C05480=1211.778,235.432,-60.754,-177.175,6.527,148.360
C05481=1211.773,235.681,-60.780,-177.172,6.529,148.360
C05482=1211.768,235.930,-60.806,-177.170,6.531,148.360
C05483=1211.764,236.179,-60.832,-177.168,6.533,148.360
C05484=1211.759,236.427,-60.857,-177.165,6.535,148.359
C05485=1211.755,236.676,-60.883,-177.163,6.537,148.359
C05486=1211.751,236.947,-60.912,-177.160,6.540,148.359
C05487=1211.745,237.218,-60.939,-177.157,6.542,148.359
C05488=1211.740,237.490,-60.968,-177.154,6.544,148.358
C05489=1211.736,237.761,-60.997,-177.151,6.546,148.358
C05490=1211.731,238.010,-61.022,-177.148,6.548,148.358
C05491=1211.727,238.258,-61.048,-177.146,6.550,148.358
C05492=1211.722,238.507,-61.074,-177.144,6.552,148.357
C05493=1211.717,238.756,-61.100,-177.141,6.554,148.357
C05494=1211.713,239.004,-61.126,-177.138,6.557,148.357
C05495=1211.709,239.253,-61.152,-177.136,6.559,148.357
C05496=1211.704,239.501,-61.178,-177.133,6.561,148.356
C05497=1211.699,239.751,-61.204,-177.131,6.563,148.356
C05498=1211.695,239.999,-61.230,-177.128,6.565,148.356
C05499=1211.691,240.247,-61.256,-177.126,6.567,148.356
C05500=1211.686,240.496,-61.282,-177.123,6.568,148.355
C05501=1211.682,240.745,-61.308,-177.120,6.571,148.355
C05502=1211.677,240.994,-61.334,-177.118,6.573,148.355
C05503=1211.673,241.242,-61.360,-177.115,6.575,148.355
C05504=1211.668,241.491,-61.387,-177.113,6.577,148.355
C05505=1211.664,241.739,-61.412,-177.110,6.579,148.354
C05506=1211.660,241.987,-61.438,-177.108,6.581,148.354
C05507=1211.655,242.236,-61.465,-177.105,6.583,148.354
C05508=1211.650,242.485,-61.491,-177.102,6.586,148.354
C05509=1211.647,242.733,-61.517,-177.100,6.588,148.353
C05510=1211.642,242.982,-61.543,-177.097,6.590,148.353
C05511=1211.637,243.230,-61.569,-177.095,6.592,148.353
C05512=1211.632,243.479,-61.596,-177.092,6.594,148.352
C05513=1211.628,243.728,-61.622,-177.090,6.596,148.352
C05514=1211.624,243.976,-61.648,-177.088,6.598,148.352
C05515=1211.619,244.225,-61.674,-177.084,6.600,148.352
C05516=1211.615,244.473,-61.701,-177.082,6.602,148.351
C05517=1211.610,244.722,-61.727,-177.080,6.604,148.351
C05518=1211.606,244.971,-61.754,-177.077,6.606,148.351
C05519=1211.602,245.219,-61.779,-177.075,6.609,148.351
C05520=1211.596,245.468,-61.805,-177.072,6.610,148.351
C05521=1211.592,245.716,-61.832,-177.069,6.613,148.350
C05522=1211.588,245.965,-61.858,-177.067,6.615,148.350
C05523=1211.584,246.213,-61.885,-177.064,6.617,148.350
C05524=1211.579,246.462,-61.912,-177.062,6.619,148.350
C05525=1211.575,246.711,-61.937,-177.060,6.621,148.350
C05526=1211.570,246.959,-61.965,-177.057,6.623,148.349
C05527=1211.566,247.208,-61.990,-177.054,6.626,148.349
C05528=1211.561,247.456,-62.017,-177.052,6.628,148.349
C05529=1211.557,247.705,-62.043,-177.049,6.630,148.349
C05530=1211.552,247.954,-62.070,-177.046,6.632,148.348
C05531=1211.548,248.202,-62.097,-177.044,6.634,148.348
C05532=1211.543,248.451,-62.123,-177.041,6.636,148.348
C05533=1211.540,248.699,-62.149,-177.039,6.639,148.348
C05534=1211.535,248.948,-62.176,-177.036,6.641,148.348
C05535=1211.531,249.196,-62.202,-177.034,6.642,148.347
C05536=1211.526,249.445,-62.229,-177.032,6.645,148.347
C05537=1211.521,249.693,-62.255,-177.029,6.646,148.347
C05538=1211.516,249.941,-62.282,-177.026,6.649,148.347
C05539=1211.512,250.190,-62.309,-177.024,6.651,148.346
C05540=1211.508,250.438,-62.335,-177.021,6.653,148.346
C05541=1211.503,250.687,-62.362,-177.019,6.655,148.346
C05542=1211.499,250.935,-62.388,-177.016,6.657,148.346
C05543=1211.494,251.184,-62.415,-177.013,6.660,148.345
C05544=1211.490,251.432,-62.442,-177.011,6.662,148.345
C05545=1211.486,251.682,-62.468,-177.008,6.664,148.345
C05546=1211.481,251.930,-62.495,-177.006,6.666,148.345
C05547=1211.478,252.179,-62.522,-177.003,6.669,148.345
C05548=1211.473,252.427,-62.549,-177.000,6.671,148.344
C05549=1211.468,252.676,-62.576,-176.998,6.673,148.344
C05550=1211.464,252.924,-62.602,-176.996,6.675,148.344
C05551=1211.459,253.173,-62.629,-176.993,6.677,148.344
C05552=1211.455,253.421,-62.656,-176.990,6.680,148.344
C05553=1211.450,253.670,-62.683,-176.988,6.682,148.344
C05554=1211.446,253.918,-62.709,-176.986,6.684,148.343
C05555=1211.441,254.167,-62.736,-176.983,6.686,148.343
C05556=1211.437,254.415,-62.763,-176.981,6.688,148.343
C05557=1211.433,254.664,-62.789,-176.978,6.690,148.343
C05558=1211.428,254.912,-62.816,-176.975,6.693,148.342
C05559=1211.423,255.161,-62.843,-176.973,6.694,148.342
C05560=1211.419,255.409,-62.870,-176.971,6.697,148.342
C05561=1211.415,255.658,-62.897,-176.968,6.699,148.342
C05562=1211.411,255.907,-62.924,-176.965,6.701,148.342
C05563=1211.406,256.155,-62.951,-176.963,6.703,148.341
C05564=1211.401,256.404,-62.978,-176.960,6.705,148.341
C05565=1211.397,256.652,-63.005,-176.957,6.708,148.341
C05566=1211.393,256.900,-63.032,-176.955,6.710,148.341
C05567=1211.388,257.149,-63.059,-176.953,6.712,148.341
C05568=1211.383,257.397,-63.086,-176.950,6.714,148.340
C05569=1211.379,257.646,-63.113,-176.947,6.717,148.340
C05570=1211.375,257.894,-63.140,-176.945,6.719,148.340
C05571=1211.371,258.143,-63.167,-176.942,6.721,148.340
C05572=1211.366,258.391,-63.195,-176.940,6.723,148.340
C05573=1211.362,258.640,-63.222,-176.937,6.726,148.339
C05574=1211.357,258.888,-63.249,-176.935,6.728,148.339
C05575=1211.352,259.137,-63.276,-176.932,6.730,148.339
C05576=1211.349,259.385,-63.302,-176.930,6.732,148.339
C05577=1211.344,259.634,-63.330,-176.927,6.735,148.339
C05578=1211.340,259.883,-63.357,-176.925,6.737,148.339
C05579=1211.335,260.131,-63.384,-176.922,6.739,148.338
C05580=1211.331,260.379,-63.412,-176.920,6.741,148.338
C05581=1211.326,260.627,-63.439,-176.917,6.744,148.338
C05582=1211.321,260.876,-63.466,-176.915,6.746,148.338
C05583=1211.317,261.125,-63.493,-176.912,6.748,148.338
C05584=1211.313,261.374,-63.520,-176.910,6.750,148.337
C05585=1211.308,261.621,-63.548,-176.907,6.753,148.337
C05586=1211.305,261.870,-63.575,-176.904,6.755,148.337
C05587=1211.300,262.118,-63.602,-176.902,6.757,148.337
C05588=1211.296,262.367,-63.629,-176.899,6.760,148.337
C05589=1211.291,262.615,-63.657,-176.897,6.762,148.336
C05590=1211.286,262.888,-63.687,-176.894,6.763,148.336
C05591=1211.281,263.161,-63.716,-176.891,6.766,148.336
C05592=1211.277,263.434,-63.747,-176.888,6.769,148.336
C05593=1211.272,263.706,-63.777,-176.886,6.771,148.336
C05594=1211.268,263.954,-63.804,-176.883,6.774,148.336
C05595=1211.263,264.203,-63.831,-176.881,6.776,148.335
C05596=1211.259,264.452,-63.859,-176.878,6.778,148.335
C05597=1211.254,264.700,-63.887,-176.876,6.780,148.335
C05598=1211.249,264.949,-63.914,-176.873,6.783,148.335
C05599=1211.245,265.197,-63.941,-176.871,6.785,148.335
C05600=1211.241,265.446,-63.970,-176.868,6.787,148.334
C05601=1211.236,265.694,-63.997,-176.865,6.790,148.334
C05602=1211.232,265.942,-64.024,-176.863,6.792,148.334
C05603=1211.227,266.191,-64.051,-176.861,6.794,148.334
C05604=1211.224,266.439,-64.080,-176.857,6.797,148.334
C05605=1211.219,266.688,-64.107,-176.855,6.799,148.334
C05606=1211.215,266.936,-64.134,-176.853,6.801,148.333
C05607=1211.210,267.185,-64.162,-176.850,6.804,148.333
C05608=1211.206,267.433,-64.190,-176.848,6.806,148.333
C05609=1211.201,267.681,-64.217,-176.845,6.808,148.333
C05610=1211.197,267.930,-64.245,-176.843,6.810,148.333
C05611=1211.192,268.179,-64.272,-176.840,6.813,148.333
C05612=1211.188,268.426,-64.300,-176.838,6.815,148.333
C05613=1211.184,268.676,-64.328,-176.835,6.817,148.332
C05614=1211.180,268.923,-64.355,-176.832,6.820,148.332
C05615=1211.175,269.172,-64.383,-176.830,6.822,148.332
C05616=1211.170,269.421,-64.411,-176.828,6.824,148.332
C05617=1211.166,269.669,-64.439,-176.825,6.827,148.332
C05618=1211.161,269.917,-64.466,-176.822,6.829,148.331
C05619=1211.158,270.166,-64.494,-176.820,6.831,148.331
C05620=1211.153,270.414,-64.522,-176.817,6.834,148.331
C05621=1211.148,270.662,-64.550,-176.815,6.836,148.331
C05622=1211.144,270.911,-64.578,-176.812,6.838,148.331
C05623=1211.140,271.159,-64.606,-176.810,6.841,148.331
C05624=1211.135,271.407,-64.633,-176.808,6.843,148.331
C05625=1211.131,271.656,-64.661,-176.805,6.845,148.330
C05626=1211.126,271.904,-64.689,-176.802,6.848,148.330
C05627=1211.122,272.153,-64.717,-176.800,6.850,148.330
C05628=1211.118,272.401,-64.744,-176.797,6.852,148.330
C05629=1211.113,272.649,-64.773,-176.795,6.855,148.330
C05630=1211.109,272.898,-64.801,-176.792,6.857,148.330
C05631=1211.104,273.147,-64.828,-176.790,6.859,148.330
C05632=1211.101,273.395,-64.856,-176.787,6.862,148.329
C05633=1211.096,273.643,-64.884,-176.785,6.864,148.329
C05634=1211.092,273.892,-64.913,-176.782,6.867,148.329
C05635=1211.087,274.140,-64.940,-176.779,6.869,148.329
C05636=1211.082,274.388,-64.969,-176.777,6.871,148.329
C05637=1211.078,274.637,-64.996,-176.775,6.874,148.329
C05638=1211.074,274.885,-65.024,-176.772,6.876,148.328
C05639=1211.070,275.134,-65.053,-176.770,6.878,148.328
C05640=1211.065,275.382,-65.080,-176.767,6.881,148.328
C05641=1211.061,275.630,-65.109,-176.765,6.883,148.328
C05642=1211.056,275.879,-65.137,-176.762,6.885,148.328
C05643=1211.053,276.127,-65.165,-176.759,6.888,148.328
C05644=1211.048,276.375,-65.193,-176.757,6.890,148.328
C05645=1211.044,276.624,-65.222,-176.754,6.893,148.328
C05646=1211.039,276.872,-65.249,-176.752,6.895,148.327
C05647=1211.035,277.121,-65.278,-176.750,6.897,148.327
C05648=1211.031,277.368,-65.306,-176.747,6.900,148.327
C05649=1211.026,277.617,-65.335,-176.744,6.902,148.327
C05650=1211.022,277.865,-65.362,-176.742,6.904,148.327
C05651=1211.018,278.114,-65.391,-176.739,6.907,148.327
C05652=1211.013,278.362,-65.419,-176.737,6.909,148.327
C05653=1211.009,278.611,-65.447,-176.734,6.912,148.327
C05654=1211.004,278.859,-65.475,-176.732,6.914,148.326
C05655=1211.000,279.107,-65.504,-176.730,6.916,148.326
C05656=1210.995,279.356,-65.532,-176.727,6.919,148.326
C05657=1210.991,279.604,-65.560,-176.725,6.922,148.326
C05658=1210.986,279.852,-65.589,-176.722,6.924,148.326
C05659=1210.983,280.101,-65.617,-176.719,6.927,148.326
C05660=1210.978,280.350,-65.645,-176.717,6.929,148.326
C05661=1210.974,280.598,-65.673,-176.714,6.931,148.325
C05662=1210.970,280.846,-65.703,-176.712,6.934,148.325
C05663=1210.965,281.094,-65.730,-176.709,6.937,148.325
C05664=1210.961,281.343,-65.759,-176.707,6.939,148.325
C05665=1210.956,281.591,-65.787,-176.705,6.941,148.325
C05666=1210.952,281.839,-65.816,-176.702,6.944,148.325
C05667=1210.948,282.088,-65.844,-176.699,6.946,148.325
C05668=1210.943,282.336,-65.873,-176.697,6.949,148.325
C05669=1210.939,282.584,-65.902,-176.695,6.951,148.325
C05670=1210.935,282.832,-65.929,-176.692,6.953,148.325
C05671=1210.930,283.081,-65.958,-176.689,6.956,148.324
C05672=1210.927,283.329,-65.987,-176.687,6.958,148.324
C05673=1210.922,283.577,-66.015,-176.684,6.961,148.324
C05674=1210.917,283.826,-66.044,-176.682,6.963,148.324
C05675=1210.913,284.074,-66.072,-176.679,6.966,148.324
C05676=1210.908,284.322,-66.101,-176.677,6.968,148.324
C05677=1210.904,284.571,-66.130,-176.675,6.970,148.324
C05678=1210.900,284.819,-66.158,-176.672,6.973,148.323
C05679=1210.895,285.067,-66.187,-176.670,6.975,148.323
C05680=1210.891,285.316,-66.216,-176.667,6.978,148.323
C05681=1210.887,285.564,-66.245,-176.665,6.980,148.323
C05682=1210.882,285.812,-66.273,-176.662,6.982,148.323
C05683=1210.878,286.061,-66.302,-176.659,6.985,148.323
C05684=1210.874,286.309,-66.330,-176.657,6.988,148.323
C05685=1210.869,286.558,-66.359,-176.655,6.991,148.323
C05686=1210.865,286.806,-66.389,-176.652,6.992,148.323
C05687=1210.861,287.054,-66.416,-176.649,6.995,148.323
C05688=1210.856,287.303,-66.445,-176.647,6.998,148.323
C05689=1210.852,287.551,-66.475,-176.645,7.001,148.323
C05690=1210.847,287.799,-66.503,-176.642,7.003,148.322
C05691=1210.844,288.047,-66.532,-176.640,7.005,148.322
C05692=1210.839,288.296,-66.561,-176.637,7.008,148.322
C05693=1210.834,288.543,-66.590,-176.635,7.010,148.322
C05694=1210.830,288.818,-66.622,-176.632,7.013,148.322
C05695=1210.825,289.093,-66.653,-176.629,7.016,148.322
C05696=1210.821,289.367,-66.686,-176.626,7.019,148.322
C05697=1210.816,289.641,-66.717,-176.624,7.022,148.322
C05698=1210.811,289.888,-66.746,-176.621,7.024,148.321
C05699=1210.807,290.137,-66.775,-176.619,7.026,148.321
C05700=1210.803,290.386,-66.805,-176.616,7.029,148.321
C05701=1210.798,290.635,-66.833,-176.614,7.031,148.321
C05702=1210.793,290.882,-66.862,-176.612,7.034,148.321
C05703=1210.790,291.130,-66.891,-176.609,7.036,148.321
C05704=1210.785,291.379,-66.920,-176.606,7.039,148.321
C05705=1210.781,291.627,-66.950,-176.604,7.041,148.321
C05706=1210.776,291.875,-66.979,-176.601,7.044,148.321
C05707=1210.772,292.124,-67.007,-176.599,7.046,148.321
C05708=1210.768,292.372,-67.037,-176.597,7.049,148.321
C05709=1210.764,292.620,-67.066,-176.594,7.051,148.321
C05710=1210.759,292.868,-67.096,-176.591,7.054,148.321
C05711=1210.755,293.116,-67.123,-176.589,7.057,148.320
C05712=1210.751,293.365,-67.153,-176.587,7.059,148.320
C05713=1210.747,293.613,-67.182,-176.584,7.062,148.320
C05714=1210.743,293.861,-67.212,-176.582,7.064,148.320
C05715=1210.738,294.110,-67.241,-176.579,7.067,148.320
C05716=1210.733,294.358,-67.270,-176.577,7.069,148.320
C05717=1210.729,294.606,-67.299,-176.574,7.072,148.320
C05718=1210.725,294.854,-67.329,-176.572,7.074,148.320
C05719=1210.721,295.102,-67.358,-176.570,7.077,148.320
C05720=1210.716,295.351,-67.387,-176.567,7.079,148.320
C05721=1210.712,295.600,-67.416,-176.565,7.082,148.320
C05722=1210.707,295.847,-67.445,-176.563,7.085,148.320
C05723=1210.703,296.095,-67.475,-176.559,7.087,148.320
C05724=1210.699,296.344,-67.504,-176.557,7.090,148.319
C05725=1210.695,296.592,-67.534,-176.555,7.093,148.319
C05726=1210.691,296.840,-67.563,-176.553,7.095,148.319
C05727=1210.686,297.088,-67.593,-176.550,7.098,148.319
C05728=1210.682,297.337,-67.622,-176.548,7.100,148.319
C05729=1210.678,297.585,-67.651,-176.545,7.103,148.319
C05730=1210.673,297.833,-67.681,-176.543,7.105,148.319
C05731=1210.669,298.081,-67.710,-176.540,7.108,148.319
C05732=1210.665,298.329,-67.739,-176.538,7.110,148.319
C05733=1210.661,298.577,-67.769,-176.535,7.114,148.319
C05734=1210.657,298.826,-67.798,-176.533,7.115,148.319
C05735=1210.652,299.074,-67.828,-176.530,7.118,148.319
C05736=1210.647,299.322,-67.858,-176.528,7.121,148.319
C05737=1210.643,299.571,-67.887,-176.525,7.124,148.319
C05738=1210.639,299.819,-67.917,-176.523,7.126,148.319
C05739=1210.635,300.067,-67.946,-176.521,7.129,148.319
C05740=1210.631,300.316,-67.976,-176.518,7.131,148.319
C05741=1210.627,300.564,-68.005,-176.516,7.134,148.319
C05742=1210.621,300.812,-68.035,-176.514,7.136,148.319
C05743=1210.617,301.060,-68.064,-176.511,7.139,148.319
C05744=1210.613,301.308,-68.094,-176.509,7.142,148.319
C05745=1210.609,301.556,-68.124,-176.506,7.145,148.318
C05746=1210.605,301.804,-68.153,-176.504,7.147,148.318
C05747=1210.600,302.052,-68.183,-176.501,7.150,148.318
C05748=1210.595,302.301,-68.213,-176.499,7.152,148.318
C05749=1210.591,302.549,-68.242,-176.496,7.155,148.318
C05750=1210.587,302.798,-68.272,-176.494,7.157,148.318
C05751=1210.583,303.045,-68.302,-176.492,7.160,148.318
C05752=1210.579,303.293,-68.331,-176.490,7.162,148.318
C05753=1210.574,303.542,-68.361,-176.487,7.166,148.318
C05754=1210.570,303.790,-68.391,-176.485,7.168,148.318
C05755=1210.566,304.038,-68.421,-176.482,7.171,148.318
C05756=1210.561,304.287,-68.451,-176.480,7.173,148.318
C05757=1210.557,304.535,-68.481,-176.477,7.176,148.318
C05758=1210.553,304.782,-68.511,-176.475,7.178,148.318
C05759=1210.549,305.031,-68.540,-176.472,7.181,148.318
C05760=1210.544,305.279,-68.570,-176.470,7.184,148.318
C05761=1210.540,305.528,-68.600,-176.468,7.186,148.318
C05762=1210.536,305.775,-68.630,-176.465,7.189,148.318
C05763=1210.531,306.024,-68.660,-176.463,7.192,148.318
C05764=1210.527,306.271,-68.690,-176.460,7.195,148.318
C05765=1210.523,306.520,-68.720,-176.458,7.197,148.318
C05766=1210.518,306.768,-68.750,-176.455,7.200,148.318
C05767=1210.514,307.016,-68.780,-176.453,7.202,148.318
C05768=1210.510,307.264,-68.809,-176.451,7.205,148.318
C05769=1210.506,307.513,-68.840,-176.448,7.207,148.318
C05770=1210.502,307.761,-68.870,-176.446,7.210,148.318
C05771=1210.497,308.009,-68.901,-176.444,7.213,148.318
C05772=1210.493,308.257,-68.930,-176.441,7.216,148.318
C05773=1210.489,308.506,-68.959,-176.439,7.218,148.318
C05774=1210.484,308.754,-68.990,-176.437,7.221,148.318
C05775=1210.480,309.002,-69.020,-176.434,7.224,148.318
C05776=1210.475,309.250,-69.050,-176.432,7.226,148.318
C05777=1210.472,309.497,-69.081,-176.429,7.229,148.318
C05778=1210.467,309.746,-69.110,-176.427,7.232,148.318
C05779=1210.463,309.994,-69.141,-176.424,7.235,148.318
C05780=1210.459,310.243,-69.171,-176.422,7.237,148.318
C05781=1210.455,310.491,-69.201,-176.420,7.240,148.318
C05782=1210.450,310.739,-69.231,-176.418,7.242,148.318
C05783=1210.446,310.987,-69.262,-176.415,7.246,148.318
C05784=1210.442,311.234,-69.292,-176.413,7.248,148.318
C05785=1210.437,311.483,-69.322,-176.410,7.251,148.318
C05786=1210.433,311.731,-69.352,-176.408,7.254,148.318
C05787=1210.428,311.979,-69.382,-176.406,7.256,148.318
C05788=1210.425,312.228,-69.413,-176.403,7.259,148.318
C05789=1210.420,312.476,-69.443,-176.401,7.262,148.318
C05790=1210.416,312.723,-69.474,-176.399,7.265,148.318
C05791=1210.411,312.972,-69.504,-176.397,7.267,148.318
C05792=1210.408,313.219,-69.534,-176.394,7.270,148.318
C05793=1210.403,313.467,-69.564,-176.392,7.272,148.318
C05794=1210.399,313.716,-69.594,-176.389,7.275,148.318
C05795=1210.395,313.964,-69.625,-176.387,7.278,148.318
C05796=1210.390,314.212,-69.656,-176.385,7.281,148.318
C05797=1210.386,314.460,-69.686,-176.382,7.284,148.318
C05798=1210.381,314.736,-69.720,-176.379,7.287,148.318
C05799=1210.376,315.012,-69.754,-176.377,7.289,148.318
C05800=1210.371,315.289,-69.787,-176.375,7.292,148.318
C05801=1210.368,315.565,-69.821,-176.372,7.295,148.318
C05802=1210.363,315.813,-69.852,-176.370,7.298,148.318
C05803=1210.359,316.061,-69.883,-176.367,7.301,148.318
C05804=1210.355,316.308,-69.913,-176.365,7.304,148.318
C05805=1210.351,316.558,-69.944,-176.362,7.307,148.318
C05806=1210.346,316.806,-69.974,-176.361,7.309,148.318
C05807=1210.342,317.053,-70.005,-176.358,7.312,148.318
C05808=1210.337,317.301,-70.035,-176.356,7.314,148.318
C05809=1210.333,317.550,-70.066,-176.353,7.317,148.318
C05810=1210.330,317.797,-70.097,-176.351,7.320,148.318
C05811=1210.325,318.045,-70.127,-176.349,7.323,148.318
C05812=1210.320,318.293,-70.158,-176.346,7.326,148.318
C05813=1210.317,318.542,-70.189,-176.344,7.328,148.318
C05814=1210.312,318.790,-70.219,-176.342,7.332,148.318
C05815=1210.308,319.038,-70.250,-176.340,7.334,148.318
C05816=1210.303,319.286,-70.281,-176.337,7.337,148.318
C05817=1210.300,319.534,-70.311,-176.335,7.339,148.318
C05818=1210.295,319.782,-70.342,-176.333,7.342,148.318
C05819=1210.291,320.030,-70.373,-176.330,7.345,148.318
C05820=1210.287,320.278,-70.404,-176.328,7.348,148.319
C05821=1210.283,320.526,-70.434,-176.326,7.351,148.319
C05822=1210.278,320.774,-70.465,-176.324,7.353,148.319
C05823=1210.274,321.023,-70.496,-176.321,7.356,148.319
C05824=1210.270,321.271,-70.527,-176.319,7.359,148.319
C05825=1210.266,321.518,-70.557,-176.317,7.362,148.319
C05826=1210.262,321.766,-70.589,-176.314,7.364,148.319
C05827=1210.257,322.014,-70.620,-176.312,7.367,148.319
C05828=1210.253,322.262,-70.650,-176.310,7.370,148.319
C05829=1210.249,322.511,-70.682,-176.308,7.373,148.319
C05830=1210.244,322.759,-70.712,-176.305,7.376,148.319
C05831=1210.240,323.007,-70.743,-176.303,7.378,148.319
C05832=1210.237,323.255,-70.774,-176.301,7.381,148.319
C05833=1210.232,323.503,-70.805,-176.299,7.384,148.319
C05834=1210.227,323.751,-70.836,-176.296,7.387,148.319
C05835=1210.223,323.999,-70.867,-176.294,7.390,148.319
C05836=1210.219,324.247,-70.899,-176.292,7.392,148.319
C05837=1210.215,324.495,-70.930,-176.290,7.396,148.320
C05838=1210.211,324.743,-70.960,-176.287,7.398,148.319
C05839=1210.206,324.991,-70.991,-176.285,7.401,148.319
C05840=1210.203,325.239,-71.022,-176.283,7.403,148.320
C05841=1210.198,325.487,-71.053,-176.280,7.406,148.320
C05842=1210.194,325.735,-71.084,-176.278,7.410,148.320
C05843=1210.190,325.983,-71.116,-176.276,7.412,148.320
C05844=1210.186,326.231,-71.147,-176.274,7.415,148.320
C05845=1210.181,326.479,-71.178,-176.272,7.417,148.320
C05846=1210.177,326.727,-71.209,-176.269,7.420,148.320
C05847=1210.173,326.975,-71.240,-176.267,7.423,148.320
C05848=1210.168,327.223,-71.271,-176.265,7.426,148.320
C05849=1210.165,327.471,-71.303,-176.263,7.429,148.320
C05850=1210.160,327.719,-71.334,-176.260,7.432,148.320
C05851=1210.156,327.967,-71.366,-176.258,7.435,148.321
C05852=1210.152,328.215,-71.396,-176.256,7.437,148.321
C05853=1210.147,328.463,-71.428,-176.254,7.440,148.321
C05854=1210.143,328.711,-71.459,-176.252,7.443,148.321
C05855=1210.139,328.959,-71.490,-176.250,7.446,148.321
C05856=1210.135,329.207,-71.522,-176.247,7.449,148.321
C05857=1210.130,329.455,-71.552,-176.245,7.452,148.321
C05858=1210.127,329.703,-71.584,-176.243,7.455,148.321
C05859=1210.122,329.951,-71.615,-176.241,7.457,148.321
C05860=1210.118,330.199,-71.647,-176.238,7.460,148.321
C05861=1210.114,330.447,-71.678,-176.237,7.463,148.321
C05862=1210.110,330.695,-71.709,-176.234,7.466,148.321
C05863=1210.106,330.943,-71.741,-176.232,7.469,148.322
C05864=1210.102,331.191,-71.772,-176.230,7.472,148.322
C05865=1210.097,331.439,-71.804,-176.227,7.475,148.322
C05866=1210.093,331.688,-71.835,-176.226,7.477,148.322
C05867=1210.088,331.935,-71.867,-176.223,7.480,148.322
C05868=1210.085,332.183,-71.898,-176.221,7.483,148.322
C05869=1210.080,332.431,-71.929,-176.219,7.486,148.322
C05870=1210.076,332.679,-71.961,-176.217,7.489,148.322
C05871=1210.072,332.926,-71.993,-176.215,7.492,148.323
C05872=1210.068,333.175,-72.024,-176.212,7.495,148.323
C05873=1210.064,333.423,-72.056,-176.211,7.497,148.323
C05874=1210.059,333.671,-72.088,-176.208,7.500,148.323
C05875=1210.055,333.919,-72.119,-176.206,7.503,148.323
C05876=1210.051,334.167,-72.150,-176.204,7.506,148.323
C05877=1210.047,334.415,-72.182,-176.201,7.509,148.323
C05878=1210.042,334.662,-72.214,-176.200,7.512,148.323
C05879=1210.038,334.911,-72.245,-176.198,7.515,148.324
C05880=1210.034,335.158,-72.277,-176.195,7.517,148.324
C05881=1210.030,335.406,-72.309,-176.193,7.521,148.324
C05882=1210.026,335.654,-72.340,-176.192,7.523,148.324
C05883=1210.021,335.903,-72.372,-176.189,7.526,148.324
C05884=1210.017,336.151,-72.404,-176.187,7.529,148.324
C05885=1210.013,336.398,-72.435,-176.185,7.532,148.324
C05886=1210.009,336.646,-72.467,-176.182,7.535,148.324
C05887=1210.005,336.894,-72.499,-176.181,7.537,148.325
C05888=1210.001,337.142,-72.531,-176.178,7.541,148.325
C05889=1209.997,337.390,-72.563,-176.177,7.543,148.325
C05890=1209.992,337.639,-72.594,-176.174,7.546,148.325
C05891=1209.988,337.886,-72.626,-176.172,7.549,148.325
C05892=1209.984,338.134,-72.658,-176.170,7.552,148.325
C05893=1209.980,338.382,-72.689,-176.168,7.555,148.325
C05894=1209.975,338.630,-72.722,-176.166,7.558,148.326
C05895=1209.972,338.878,-72.754,-176.164,7.561,148.326
C05896=1209.967,339.125,-72.785,-176.162,7.564,148.326
C05897=1209.963,339.374,-72.817,-176.160,7.567,148.326
C05898=1209.959,339.622,-72.849,-176.158,7.569,148.326
C05899=1209.955,339.869,-72.881,-176.156,7.573,148.326
C05900=1209.951,340.117,-72.913,-176.153,7.576,148.327
C05901=1209.947,340.365,-72.945,-176.152,7.578,148.327
C05902=1209.942,340.643,-72.981,-176.149,7.581,148.327
C05903=1209.937,340.921,-73.016,-176.147,7.585,148.327
C05904=1209.933,341.200,-73.053,-176.145,7.588,148.327
C05905=1209.928,341.478,-73.089,-176.142,7.592,148.327
C05906=1209.924,341.726,-73.121,-176.140,7.595,148.328
C05907=1209.919,341.973,-73.153,-176.139,7.597,148.328
C05908=1209.915,342.222,-73.185,-176.136,7.600,148.328
C05909=1209.911,342.470,-73.217,-176.134,7.603,148.328
C05910=1209.906,342.717,-73.249,-176.132,7.606,148.328
C05911=1209.903,342.965,-73.280,-176.130,7.609,148.328
C05912=1209.899,343.213,-73.314,-176.128,7.612,148.329
C05913=1209.894,343.460,-73.345,-176.127,7.615,148.329
C05914=1209.890,343.709,-73.378,-176.124,7.618,148.329
C05915=1209.886,343.957,-73.409,-176.122,7.621,148.329
C05916=1209.882,344.205,-73.442,-176.120,7.624,148.329
C05917=1209.877,344.452,-73.473,-176.118,7.627,148.329
C05918=1209.873,344.700,-73.506,-176.116,7.629,148.330
C05919=1209.869,344.948,-73.538,-176.114,7.633,148.330
C05920=1209.865,345.196,-73.571,-176.112,7.635,148.330
C05921=1209.861,345.444,-73.602,-176.110,7.639,148.330
C05922=1209.857,345.692,-73.635,-176.108,7.641,148.330
C05923=1209.853,345.940,-73.667,-176.106,7.645,148.331
C05924=1209.848,346.188,-73.700,-176.105,7.647,148.331
C05925=1209.843,346.436,-73.732,-176.102,7.650,148.331
C05926=1209.840,346.683,-73.764,-176.101,7.653,148.331
C05927=1209.836,346.931,-73.797,-176.098,7.656,148.331
C05928=1209.832,347.179,-73.829,-176.096,7.660,148.332
C05929=1209.828,347.427,-73.862,-176.095,7.662,148.332
C05930=1209.823,347.674,-73.893,-176.092,7.665,148.332
C05931=1209.819,347.923,-73.926,-176.091,7.668,148.332
C05932=1209.815,348.171,-73.959,-176.089,7.671,148.332
C05933=1209.811,348.419,-73.991,-176.087,7.674,148.333
C05934=1209.807,348.666,-74.024,-176.085,7.677,148.333
C05935=1209.802,348.914,-74.056,-176.083,7.680,148.333
C05936=1209.798,349.162,-74.088,-176.081,7.683,148.333
C05937=1209.794,349.410,-74.121,-176.079,7.686,148.333
C05938=1209.790,349.658,-74.153,-176.077,7.689,148.334
C05939=1209.786,349.905,-74.186,-176.076,7.692,148.334
C05940=1209.781,350.153,-74.218,-176.074,7.695,148.334
C05941=1209.778,350.401,-74.251,-176.072,7.698,148.334
C05942=1209.773,350.649,-74.283,-176.070,7.701,148.335
C05943=1209.769,350.897,-74.316,-176.068,7.703,148.335
C05944=1209.766,351.145,-74.348,-176.066,7.707,148.335
C05945=1209.761,351.392,-74.381,-176.064,7.709,148.335
C05946=1209.757,351.641,-74.414,-176.062,7.713,148.336
C05947=1209.752,351.888,-74.446,-176.061,7.715,148.336
C05948=1209.748,352.136,-74.478,-176.059,7.719,148.336
C05949=1209.744,352.384,-74.511,-176.057,7.721,148.336
C05950=1209.740,352.632,-74.544,-176.055,7.725,148.337
C05951=1209.737,352.879,-74.576,-176.053,7.727,148.337
C05952=1209.732,353.127,-74.610,-176.051,7.731,148.337
C05953=1209.728,353.375,-74.642,-176.050,7.733,148.337
C05954=1209.724,353.623,-74.675,-176.047,7.737,148.338
C05955=1209.719,353.871,-74.708,-176.046,7.739,148.338
C05956=1209.715,354.118,-74.740,-176.044,7.743,148.338
C05957=1209.711,354.366,-74.773,-176.042,7.745,148.338
C05958=1209.707,354.614,-74.805,-176.040,7.749,148.339
C05959=1209.703,354.862,-74.839,-176.039,7.751,148.339
C05960=1209.699,355.109,-74.871,-176.037,7.755,148.339
C05961=1209.695,355.358,-74.904,-176.035,7.757,148.339
C05962=1209.691,355.606,-74.937,-176.033,7.761,148.340
C05963=1209.687,355.853,-74.970,-176.031,7.763,148.340
C05964=1209.682,356.101,-75.003,-176.030,7.767,148.340
C05965=1209.678,356.349,-75.035,-176.028,7.769,148.340
C05966=1209.675,356.597,-75.068,-176.026,7.773,148.341
C05967=1209.670,356.844,-75.101,-176.024,7.776,148.341
C05968=1209.666,357.092,-75.134,-176.022,7.779,148.341
C05969=1209.662,357.341,-75.167,-176.021,7.781,148.341
C05970=1209.658,357.588,-75.200,-176.019,7.785,148.342
C05971=1209.654,357.836,-75.233,-176.017,7.788,148.342
C05972=1209.649,358.084,-75.266,-176.015,7.791,148.343
C05973=1209.646,358.331,-75.299,-176.014,7.794,148.343
C05974=1209.642,358.580,-75.331,-176.012,7.797,148.343
C05975=1209.637,358.827,-75.364,-176.010,7.800,148.343
C05976=1209.633,359.074,-75.397,-176.008,7.803,148.344
C05977=1209.629,359.322,-75.430,-176.007,7.806,148.344
C05978=1209.624,359.570,-75.463,-176.005,7.809,148.344
C05979=1209.620,359.817,-75.497,-176.003,7.812,148.344
C05980=1209.616,360.065,-75.530,-176.002,7.815,148.345
C05981=1209.613,360.314,-75.563,-176.000,7.818,148.345
C05982=1209.608,360.561,-75.596,-175.999,7.821,148.345
C05983=1209.604,360.810,-75.629,-175.996,7.824,148.346
C05984=1209.600,361.057,-75.662,-175.995,7.827,148.346
C05985=1209.596,361.305,-75.695,-175.993,7.830,148.346
C05986=1209.592,361.553,-75.728,-175.992,7.833,148.347
C05987=1209.587,361.801,-75.762,-175.990,7.836,148.347
C05988=1209.584,362.048,-75.794,-175.988,7.839,148.347
C05989=1209.580,362.296,-75.827,-175.987,7.842,148.348
C05990=1209.576,362.543,-75.860,-175.985,7.846,148.348
C05991=1209.572,362.791,-75.894,-175.984,7.848,148.348
C05992=1209.567,363.039,-75.927,-175.982,7.851,148.348
C05993=1209.563,363.287,-75.960,-175.980,7.855,148.349
C05994=1209.558,363.535,-75.994,-175.979,7.857,148.349
C05995=1209.555,363.782,-76.027,-175.977,7.861,148.350
C05996=1209.551,364.030,-76.061,-175.976,7.863,148.350
C05997=1209.546,364.277,-76.094,-175.974,7.866,148.350
C05998=1209.542,364.525,-76.127,-175.972,7.870,148.351
C05999=1209.538,364.773,-76.160,-175.971,7.872,148.351
C06000=1209.535,365.021,-76.194,-175.969,7.875,148.351
C06001=1209.530,365.269,-76.227,-175.968,7.879,148.352
C06002=1209.526,365.517,-76.260,-175.966,7.881,148.352
C06003=1209.522,365.764,-76.293,-175.965,7.884,148.352
C06004=1209.518,366.011,-76.327,-175.963,7.888,148.353
C06005=1209.514,366.259,-76.360,-175.962,7.890,148.353
C06006=1209.509,366.540,-76.398,-175.960,7.894,148.353
C06007=1209.505,366.820,-76.435,-175.958,7.897,148.354
C06008=1209.501,367.100,-76.473,-175.957,7.900,148.354
C06009=1209.495,367.380,-76.511,-175.955,7.904,148.354
C06010=1209.492,367.629,-76.545,-175.954,7.907,148.355
C06011=1209.488,367.876,-76.578,-175.952,7.910,148.355
C06012=1209.483,368.124,-76.611,-175.951,7.913,148.356
C06013=1209.480,368.371,-76.645,-175.949,7.916,148.356
C06014=1209.475,368.619,-76.679,-175.947,7.919,148.356
C06015=1209.471,368.867,-76.712,-175.946,7.922,148.357
C06016=1209.466,369.115,-76.745,-175.945,7.925,148.357
C06017=1209.463,369.362,-76.779,-175.944,7.928,148.358
C06018=1209.459,369.610,-76.813,-175.942,7.931,148.358
C06019=1209.455,369.858,-76.846,-175.940,7.934,148.358
C06020=1209.450,370.105,-76.880,-175.939,7.937,148.359
C06021=1209.446,370.353,-76.913,-175.938,7.940,148.359
C06022=1209.442,370.601,-76.947,-175.936,7.943,148.359
C06023=1209.438,370.848,-76.980,-175.935,7.946,148.360
C06024=1209.435,371.096,-77.014,-175.934,7.949,148.360
C06025=1209.430,371.344,-77.048,-175.933,7.952,148.361
C06026=1209.426,371.592,-77.082,-175.931,7.954,148.361
C06027=1209.422,371.839,-77.115,-175.930,7.958,148.361
C06028=1209.418,372.087,-77.148,-175.928,7.961,148.362
C06029=1209.414,372.335,-77.183,-175.927,7.964,148.362
C06030=1209.410,372.583,-77.216,-175.926,7.966,148.363
C06031=1209.406,372.830,-77.250,-175.925,7.969,148.363
C06032=1209.402,373.078,-77.283,-175.923,7.973,148.363
C06033=1209.397,373.325,-77.317,-175.922,7.976,148.364
C06034=1209.393,373.574,-77.351,-175.921,7.979,148.364
C06035=1209.390,373.821,-77.385,-175.919,7.981,148.365
C06036=1209.385,374.069,-77.418,-175.918,7.984,148.365
C06037=1209.381,374.316,-77.452,-175.917,7.987,148.365
C06038=1209.377,374.564,-77.486,-175.916,7.990,148.366
C06039=1209.373,374.812,-77.520,-175.914,7.993,148.366
C06040=1209.369,375.059,-77.554,-175.913,7.996,148.367
C06041=1209.365,375.307,-77.587,-175.912,7.999,148.367
C06042=1209.361,375.554,-77.621,-175.911,8.002,148.368
C06043=1209.357,375.802,-77.655,-175.910,8.005,148.368
C06044=1209.353,376.050,-77.689,-175.909,8.008,148.368
C06045=1209.349,376.297,-77.722,-175.907,8.011,148.369
C06046=1209.344,376.545,-77.756,-175.906,8.013,148.369
C06047=1209.341,376.793,-77.790,-175.905,8.016,148.370
C06048=1209.336,377.041,-77.824,-175.904,8.019,148.370
C06049=1209.332,377.288,-77.858,-175.903,8.022,148.370
C06050=1209.328,377.535,-77.892,-175.902,8.025,148.371
C06051=1209.324,377.784,-77.926,-175.901,8.028,148.371
C06052=1209.320,378.031,-77.960,-175.899,8.031,148.372
C06053=1209.316,378.279,-77.993,-175.898,8.033,148.372
C06054=1209.311,378.526,-78.027,-175.897,8.037,148.373
C06055=1209.308,378.774,-78.062,-175.896,8.039,148.373
C06056=1209.303,379.022,-78.095,-175.895,8.042,148.373
C06057=1209.299,379.269,-78.129,-175.894,8.045,148.374
C06058=1209.295,379.517,-78.164,-175.893,8.048,148.374
C06059=1209.291,379.765,-78.197,-175.892,8.051,148.375
C06060=1209.287,380.012,-78.231,-175.891,8.054,148.375
C06061=1209.283,380.260,-78.266,-175.889,8.056,148.376
C06062=1209.279,380.508,-78.299,-175.889,8.060,148.376
C06063=1209.275,380.755,-78.334,-175.888,8.062,148.377
C06064=1209.271,381.003,-78.368,-175.886,8.065,148.377
C06065=1209.267,381.251,-78.402,-175.886,8.068,148.378
C06066=1209.263,381.498,-78.436,-175.884,8.071,148.378
C06067=1209.258,381.746,-78.470,-175.883,8.074,148.378
C06068=1209.255,381.994,-78.504,-175.882,8.077,148.379
C06069=1209.251,382.241,-78.537,-175.881,8.080,148.379
C06070=1209.246,382.489,-78.572,-175.880,8.083,148.380
C06071=1209.243,382.737,-78.606,-175.880,8.085,148.380
C06072=1209.239,382.984,-78.641,-175.879,8.088,148.381
C06073=1209.235,383.231,-78.674,-175.878,8.091,148.381
C06074=1209.230,383.479,-78.708,-175.877,8.094,148.382
C06075=1209.227,383.727,-78.742,-175.875,8.096,148.382
C06076=1209.222,383.974,-78.777,-175.875,8.100,148.383
C06077=1209.218,384.223,-78.812,-175.873,8.102,148.383
C06078=1209.214,384.470,-78.846,-175.873,8.105,148.384
C06079=1209.209,384.718,-78.879,-175.872,8.108,148.384
C06080=1209.206,384.965,-78.914,-175.871,8.111,148.385
C06081=1209.202,385.213,-78.948,-175.870,8.113,148.385
C06082=1209.198,385.460,-78.982,-175.869,8.117,148.386
C06083=1209.194,385.708,-79.017,-175.869,8.119,148.386
C06084=1209.190,385.955,-79.051,-175.867,8.121,148.386
C06085=1209.185,386.203,-79.085,-175.867,8.124,148.387
C06086=1209.182,386.450,-79.119,-175.866,8.127,148.387
C06087=1209.177,386.699,-79.153,-175.865,8.130,148.388
C06088=1209.173,386.946,-79.188,-175.864,8.132,148.388
C06089=1209.169,387.194,-79.222,-175.863,8.135,148.389
C06090=1209.165,387.441,-79.256,-175.862,8.138,148.389
C06091=1209.162,387.689,-79.290,-175.862,8.141,148.390
C06092=1209.157,387.936,-79.325,-175.861,8.143,148.390
C06093=1209.153,388.183,-79.359,-175.860,8.146,148.391
C06094=1209.149,388.432,-79.394,-175.860,8.149,148.391
C06095=1209.145,388.679,-79.428,-175.859,8.151,148.392
C06096=1209.141,388.927,-79.462,-175.858,8.155,148.392
C06097=1209.137,389.174,-79.497,-175.857,8.157,148.393
C06098=1209.133,389.421,-79.531,-175.856,8.160,148.393
C06099=1209.129,389.669,-79.566,-175.855,8.162,148.394
C06100=1209.125,389.917,-79.600,-175.855,8.165,148.394
C06101=1209.121,390.165,-79.634,-175.854,8.168,148.394
C06102=1209.117,390.412,-79.669,-175.853,8.171,148.395
C06103=1209.112,390.660,-79.703,-175.853,8.173,148.396
C06104=1209.109,390.907,-79.737,-175.852,8.176,148.396
C06105=1209.104,391.155,-79.772,-175.851,8.179,148.397
C06106=1209.100,391.403,-79.807,-175.850,8.181,148.397
C06107=1209.097,391.650,-79.841,-175.849,8.184,148.398
C06108=1209.093,391.898,-79.875,-175.849,8.186,148.398
C06109=1209.089,392.145,-79.909,-175.848,8.189,148.398
C06110=1209.084,392.428,-79.949,-175.847,8.192,148.399
C06111=1209.079,392.710,-79.988,-175.846,8.195,148.400
C06112=1209.075,392.992,-80.028,-175.846,8.198,148.400
C06113=1209.070,393.275,-80.067,-175.846,8.201,148.401
C06114=1209.066,393.523,-80.101,-175.844,8.203,148.401
C06115=1209.062,393.770,-80.137,-175.844,8.206,148.402
C06116=1209.058,394.017,-80.171,-175.843,8.209,148.402
C06117=1209.054,394.265,-80.205,-175.843,8.211,148.403
C06118=1209.050,394.513,-80.240,-175.842,8.214,148.403
C06119=1209.045,394.760,-80.274,-175.841,8.216,148.404
C06120=1209.042,395.008,-80.309,-175.841,8.219,148.404
C06121=1209.037,395.255,-80.343,-175.840,8.221,148.405
C06122=1209.033,395.504,-80.378,-175.839,8.224,148.405
C06123=1209.030,395.750,-80.413,-175.839,8.226,148.406
C06124=1209.026,395.998,-80.447,-175.838,8.229,148.406
C06125=1209.021,396.246,-80.482,-175.837,8.231,148.407
C06126=1209.017,396.494,-80.517,-175.837,8.235,148.407
C06127=1209.014,396.741,-80.551,-175.837,8.237,148.408
C06128=1209.010,396.988,-80.586,-175.836,8.239,148.408
C06129=1209.005,397.236,-80.621,-175.835,8.242,148.409
C06130=1209.001,397.484,-80.655,-175.835,8.244,148.409
C06131=1208.998,397.731,-80.689,-175.834,8.247,148.410
C06132=1208.994,397.979,-80.724,-175.833,8.249,148.410
C06133=1208.989,398.226,-80.759,-175.833,8.251,148.411
C06134=1208.985,398.474,-80.794,-175.832,8.255,148.411
C06135=1208.981,398.721,-80.829,-175.832,8.257,148.412
C06136=1208.978,398.969,-80.863,-175.832,8.259,148.412
C06137=1208.973,399.216,-80.898,-175.831,8.262,148.413
C06138=1208.969,399.464,-80.933,-175.830,8.264,148.413
C06139=1208.965,399.712,-80.967,-175.830,8.266,148.414
C06140=1208.962,399.959,-81.002,-175.829,8.269,148.414
C06141=1208.957,400.206,-81.037,-175.829,8.271,148.415
C06142=1208.953,400.454,-81.072,-175.828,8.274,148.415
C06143=1208.949,400.702,-81.106,-175.828,8.277,148.416
C06144=1208.945,400.950,-81.141,-175.827,8.279,148.416
C06145=1208.941,401.196,-81.175,-175.827,8.281,148.417
C06146=1208.937,401.444,-81.210,-175.826,8.284,148.417
C06147=1208.933,401.692,-81.245,-175.826,8.286,148.418
C06148=1208.929,401.939,-81.280,-175.825,8.288,148.418
C06149=1208.924,402.187,-81.315,-175.825,8.290,148.419
C06150=1208.921,402.435,-81.350,-175.824,8.294,148.419
C06151=1208.917,402.681,-81.384,-175.823,8.296,148.419
C06152=1208.913,402.929,-81.419,-175.823,8.298,148.420
C06153=1208.908,403.177,-81.453,-175.823,8.300,148.421
C06154=1208.905,403.424,-81.489,-175.822,8.303,148.421
C06155=1208.900,403.672,-81.523,-175.822,8.305,148.421
C06156=1208.896,403.920,-81.558,-175.821,8.307,148.422
C06157=1208.892,404.167,-81.593,-175.821,8.310,148.422
C06158=1208.889,404.415,-81.628,-175.821,8.312,148.423
C06159=1208.885,404.662,-81.663,-175.820,8.315,148.423
C06160=1208.881,404.909,-81.698,-175.820,8.317,148.424
C06161=1208.877,405.158,-81.733,-175.819,8.319,148.424
C06162=1208.872,405.404,-81.768,-175.819,8.321,148.425
C06163=1208.868,405.653,-81.803,-175.818,8.324,148.425
C06164=1208.864,405.899,-81.838,-175.818,8.327,148.426
C06165=1208.860,406.147,-81.873,-175.817,8.329,148.426
C06166=1208.856,406.395,-81.906,-175.817,8.331,148.427
C06167=1208.853,406.642,-81.942,-175.817,8.333,148.427
C06168=1208.849,406.890,-81.977,-175.816,8.335,148.428
C06169=1208.844,407.137,-82.012,-175.816,8.337,148.428
C06170=1208.840,407.385,-82.047,-175.816,8.340,148.429
C06171=1208.836,407.632,-82.082,-175.815,8.342,148.429
C06172=1208.832,407.880,-82.117,-175.814,8.345,148.430
C06173=1208.828,408.127,-82.151,-175.814,8.347,148.430
C06174=1208.824,408.375,-82.187,-175.813,8.349,148.431
C06175=1208.820,408.623,-82.222,-175.813,8.351,148.431
C06176=1208.816,408.870,-82.257,-175.813,8.354,148.432
C06177=1208.812,409.118,-82.291,-175.813,8.356,148.432
C06178=1208.808,409.364,-82.326,-175.812,8.358,148.432
C06179=1208.804,409.613,-82.361,-175.812,8.360,148.433
C06180=1208.801,409.860,-82.397,-175.812,8.362,148.434
C06181=1208.796,410.107,-82.431,-175.811,8.364,148.434
C06182=1208.792,410.355,-82.467,-175.811,8.367,148.434
C06183=1208.788,410.602,-82.501,-175.810,8.370,148.435
C06184=1208.784,410.850,-82.537,-175.809,8.372,148.435
C06185=1208.780,411.098,-82.572,-175.809,8.374,148.436
C06186=1208.776,411.345,-82.607,-175.809,8.376,148.436
C06187=1208.772,411.593,-82.642,-175.808,8.378,148.437
C06188=1208.768,411.840,-82.677,-175.808,8.380,148.437
C06189=1208.764,412.087,-82.712,-175.808,8.383,148.438
C06190=1208.760,412.335,-82.747,-175.807,8.385,148.438
C06191=1208.756,412.582,-82.782,-175.807,8.387,148.439
C06192=1208.752,412.830,-82.817,-175.807,8.389,148.439
C06193=1208.748,413.077,-82.852,-175.806,8.391,148.440
C06194=1208.744,413.325,-82.887,-175.806,8.393,148.440
C06195=1208.740,413.573,-82.923,-175.805,8.396,148.441
C06196=1208.736,413.820,-82.958,-175.805,8.398,148.441
C06197=1208.732,414.068,-82.993,-175.805,8.400,148.441
C06198=1208.728,414.315,-83.028,-175.804,8.402,148.442
C06199=1208.723,414.563,-83.063,-175.804,8.404,148.442
C06200=1208.720,414.810,-83.098,-175.804,8.406,148.443
C06201=1208.715,415.057,-83.133,-175.803,8.409,148.443
C06202=1208.712,415.305,-83.168,-175.803,8.411,148.444
C06203=1208.708,415.552,-83.204,-175.802,8.413,148.444
C06204=1208.703,415.800,-83.238,-175.802,8.415,148.445
C06205=1208.700,416.047,-83.274,-175.802,8.416,148.445
C06206=1208.695,416.309,-83.311,-175.801,8.419,148.446
C06207=1208.692,416.571,-83.348,-175.801,8.421,148.446
C06208=1208.690,416.833,-83.385,-175.800,8.424,148.447
C06209=1208.692,417.093,-83.422,-175.800,8.426,148.447
C06210=1208.270,417.094,-83.458,-175.803,8.436,148.451
C06211=1208.269,416.830,-83.421,-175.804,8.434,148.450
C06212=1208.270,416.565,-83.385,-175.804,8.432,148.450
C06213=1208.274,416.301,-83.347,-175.805,8.430,148.449
C06214=1208.278,416.037,-83.309,-175.805,8.427,148.449
C06215=1208.282,415.789,-83.274,-175.805,8.426,148.448
C06216=1208.286,415.541,-83.239,-175.806,8.424,148.448
C06217=1208.290,415.295,-83.203,-175.806,8.421,148.447
C06218=1208.294,415.046,-83.168,-175.806,8.419,148.447
C06219=1208.298,414.799,-83.133,-175.807,8.417,148.447
C06220=1208.302,414.551,-83.098,-175.807,8.415,148.446
C06221=1208.306,414.304,-83.063,-175.807,8.413,148.446
C06222=1208.310,414.057,-83.028,-175.808,8.411,148.445
C06223=1208.314,413.809,-82.993,-175.808,8.408,148.445
C06224=1208.318,413.562,-82.957,-175.808,8.406,148.444
C06225=1208.323,413.314,-82.923,-175.809,8.404,148.444
C06226=1208.326,413.067,-82.887,-175.809,8.402,148.443
C06227=1208.330,412.819,-82.852,-175.809,8.400,148.443
C06228=1208.334,412.572,-82.817,-175.810,8.398,148.442
C06229=1208.338,412.324,-82.782,-175.810,8.395,148.442
C06230=1208.343,412.077,-82.747,-175.811,8.393,148.441
C06231=1208.346,411.829,-82.712,-175.811,8.391,148.441
C06232=1208.350,411.581,-82.677,-175.811,8.389,148.440
C06233=1208.355,411.334,-82.642,-175.812,8.387,148.440
C06234=1208.359,411.086,-82.607,-175.812,8.385,148.440
C06235=1208.363,410.839,-82.572,-175.812,8.382,148.439
C06236=1208.366,410.592,-82.536,-175.813,8.380,148.439
C06237=1208.370,410.344,-82.501,-175.813,8.378,148.438
C06238=1208.375,410.097,-82.466,-175.814,8.375,148.438
C06239=1208.379,409.849,-82.431,-175.814,8.373,148.437
C06240=1208.383,409.602,-82.396,-175.815,8.370,148.437
C06241=1208.386,409.354,-82.362,-175.815,8.368,148.436
C06242=1208.390,409.107,-82.326,-175.815,8.366,148.436
C06243=1208.394,408.859,-82.292,-175.816,8.364,148.435
C06244=1208.398,408.612,-82.256,-175.816,8.362,148.435
C06245=1208.403,408.364,-82.222,-175.817,8.360,148.434
C06246=1208.406,408.117,-82.186,-175.817,8.357,148.434
C06247=1208.410,407.869,-82.152,-175.817,8.355,148.433
C06248=1208.415,407.621,-82.117,-175.818,8.353,148.433
C06249=1208.418,407.374,-82.082,-175.818,8.350,148.432
C06250=1208.423,407.127,-82.047,-175.819,8.348,148.432
C06251=1208.427,406.879,-82.012,-175.819,8.346,148.431
C06252=1208.431,406.632,-81.977,-175.819,8.344,148.431
C06253=1208.434,406.384,-81.942,-175.820,8.341,148.430
C06254=1208.438,406.136,-81.907,-175.820,8.339,148.430
C06255=1208.442,405.890,-81.872,-175.821,8.337,148.429
C06256=1208.446,405.641,-81.837,-175.821,8.335,148.429
C06257=1208.451,405.394,-81.803,-175.822,8.332,148.429
C06258=1208.455,405.146,-81.767,-175.822,8.330,148.428
C06259=1208.459,404.899,-81.733,-175.822,8.327,148.427
C06260=1208.463,404.652,-81.697,-175.823,8.325,148.427
C06261=1208.467,404.403,-81.662,-175.823,8.323,148.427
C06262=1208.471,404.156,-81.629,-175.824,8.320,148.426
C06263=1208.474,403.909,-81.593,-175.824,8.318,148.425
C06264=1208.479,403.661,-81.558,-175.825,8.316,148.425
C06265=1208.483,403.414,-81.523,-175.825,8.314,148.425
C06266=1208.487,403.166,-81.488,-175.825,8.311,148.424
C06267=1208.491,402.918,-81.454,-175.826,8.308,148.423
C06268=1208.495,402.672,-81.418,-175.827,8.306,148.423
C06269=1208.499,402.424,-81.384,-175.827,8.304,148.423
C06270=1208.503,402.176,-81.350,-175.827,8.302,148.422
C06271=1208.507,401.929,-81.314,-175.828,8.299,148.422
C06272=1208.511,401.681,-81.280,-175.829,8.297,148.421
C06273=1208.515,401.433,-81.245,-175.829,8.294,148.421
C06274=1208.519,401.186,-81.209,-175.829,8.292,148.420
C06275=1208.523,400.939,-81.175,-175.830,8.289,148.420
C06276=1208.527,400.691,-81.141,-175.830,8.287,148.419
C06277=1208.531,400.444,-81.105,-175.831,8.285,148.419
C06278=1208.535,400.196,-81.071,-175.832,8.282,148.418
C06279=1208.540,399.948,-81.036,-175.832,8.280,148.418
C06280=1208.543,399.700,-81.002,-175.832,8.277,148.417
C06281=1208.547,399.454,-80.967,-175.833,8.274,148.417
C06282=1208.551,399.205,-80.932,-175.834,8.272,148.416
C06283=1208.556,398.958,-80.897,-175.834,8.270,148.416
C06284=1208.560,398.710,-80.863,-175.835,8.267,148.415
C06285=1208.563,398.463,-80.828,-175.835,8.265,148.415
C06286=1208.567,398.215,-80.793,-175.836,8.263,148.414
C06287=1208.572,397.968,-80.759,-175.836,8.260,148.414
C06288=1208.576,397.720,-80.724,-175.837,8.258,148.413
C06289=1208.579,397.473,-80.689,-175.838,8.254,148.413
C06290=1208.583,397.225,-80.654,-175.838,8.252,148.412
C06291=1208.588,396.978,-80.620,-175.838,8.250,148.412
C06292=1208.592,396.730,-80.585,-175.839,8.247,148.411
C06293=1208.596,396.482,-80.551,-175.840,8.245,148.411
C06294=1208.600,396.236,-80.516,-175.840,8.242,148.410
C06295=1208.604,395.988,-80.481,-175.841,8.240,148.410
C06296=1208.608,395.740,-80.447,-175.841,8.238,148.409
C06297=1208.612,395.492,-80.412,-175.842,8.234,148.409
C06298=1208.616,395.245,-80.378,-175.843,8.232,148.408
C06299=1208.620,394.997,-80.343,-175.843,8.229,148.408
C06300=1208.624,394.750,-80.308,-175.844,8.227,148.407
C06301=1208.628,394.502,-80.274,-175.845,8.224,148.407
C06302=1208.632,394.255,-80.239,-175.845,8.222,148.406
C06303=1208.636,394.007,-80.205,-175.846,8.219,148.406
C06304=1208.641,393.759,-80.170,-175.846,8.217,148.405
C06305=1208.644,393.511,-80.136,-175.847,8.214,148.405
C06306=1208.649,393.264,-80.101,-175.848,8.212,148.404
C06307=1208.653,392.982,-80.062,-175.849,8.209,148.404
C06308=1208.658,392.699,-80.023,-175.849,8.206,148.403
C06309=1208.662,392.417,-79.983,-175.850,8.203,148.403
C06310=1208.667,392.135,-79.943,-175.851,8.199,148.402
C06311=1208.670,391.888,-79.909,-175.851,8.197,148.401
C06312=1208.674,391.639,-79.875,-175.852,8.194,148.401
C06313=1208.679,391.392,-79.840,-175.853,8.191,148.400
C06314=1208.682,391.144,-79.806,-175.854,8.189,148.400
C06315=1208.687,390.897,-79.771,-175.855,8.186,148.400
C06316=1208.691,390.649,-79.737,-175.855,8.184,148.399
C06317=1208.695,390.402,-79.703,-175.856,8.181,148.399
C06318=1208.699,390.154,-79.668,-175.857,8.178,148.398
C06319=1208.703,389.906,-79.633,-175.857,8.176,148.398
C06320=1208.707,389.659,-79.599,-175.858,8.173,148.397
C06321=1208.711,389.412,-79.565,-175.859,8.170,148.397
C06322=1208.715,389.163,-79.530,-175.860,8.168,148.396
C06323=1208.719,388.916,-79.496,-175.860,8.165,148.396
C06324=1208.723,388.668,-79.461,-175.861,8.162,148.395
C06325=1208.727,388.421,-79.428,-175.862,8.160,148.395
C06326=1208.732,388.174,-79.393,-175.863,8.157,148.394
C06327=1208.736,387.926,-79.358,-175.864,8.154,148.394
C06328=1208.739,387.678,-79.324,-175.864,8.152,148.393
C06329=1208.743,387.430,-79.290,-175.865,8.149,148.393
C06330=1208.747,387.183,-79.256,-175.866,8.146,148.392
C06331=1208.752,386.936,-79.221,-175.867,8.143,148.392
C06332=1208.756,386.688,-79.186,-175.868,8.141,148.391
C06333=1208.760,386.440,-79.153,-175.868,8.138,148.391
C06334=1208.764,386.192,-79.118,-175.870,8.135,148.390
C06335=1208.768,385.945,-79.085,-175.870,8.132,148.390
C06336=1208.772,385.697,-79.050,-175.871,8.130,148.389
C06337=1208.775,385.449,-79.016,-175.872,8.127,148.389
C06338=1208.780,385.202,-78.981,-175.873,8.124,148.389
C06339=1208.784,384.955,-78.948,-175.874,8.121,148.388
C06340=1208.788,384.707,-78.913,-175.875,8.118,148.388
C06341=1208.793,384.459,-78.879,-175.875,8.116,148.387
C06342=1208.797,384.212,-78.845,-175.876,8.113,148.387
C06343=1208.801,383.964,-78.810,-175.877,8.110,148.386
C06344=1208.804,383.716,-78.776,-175.878,8.107,148.386
C06345=1208.809,383.469,-78.742,-175.880,8.104,148.385
C06346=1208.812,383.221,-78.708,-175.880,8.101,148.385
C06347=1208.817,382.973,-78.674,-175.881,8.099,148.384
C06348=1208.821,382.726,-78.640,-175.882,8.096,148.384
C06349=1208.825,382.478,-78.605,-175.883,8.093,148.383
C06350=1208.829,382.231,-78.571,-175.884,8.090,148.383
C06351=1208.834,381.983,-78.538,-175.885,8.087,148.382
C06352=1208.837,381.735,-78.503,-175.886,8.084,148.382
C06353=1208.841,381.488,-78.469,-175.887,8.081,148.381
C06354=1208.845,381.240,-78.435,-175.888,8.078,148.381
C06355=1208.849,380.992,-78.401,-175.889,8.076,148.381
C06356=1208.853,380.745,-78.367,-175.890,8.072,148.380
C06357=1208.857,380.498,-78.333,-175.891,8.070,148.380
C06358=1208.861,380.249,-78.298,-175.892,8.067,148.379
C06359=1208.865,380.002,-78.265,-175.893,8.065,148.379
C06360=1208.870,379.754,-78.231,-175.894,8.062,148.378
C06361=1208.873,379.506,-78.196,-175.895,8.059,148.378
C06362=1208.878,379.258,-78.163,-175.896,8.056,148.377
C06363=1208.882,379.011,-78.129,-175.897,8.053,148.377
C06364=1208.886,378.764,-78.095,-175.898,8.050,148.376
C06365=1208.890,378.515,-78.061,-175.899,8.047,148.376
C06366=1208.894,378.268,-78.027,-175.901,8.045,148.376
C06367=1208.898,378.021,-77.993,-175.901,8.042,148.375
C06368=1208.902,377.773,-77.959,-175.903,8.039,148.375
C06369=1208.906,377.525,-77.925,-175.904,8.035,148.374
C06370=1208.910,377.277,-77.891,-175.906,8.032,148.374
C06371=1208.914,377.030,-77.858,-175.907,8.029,148.373
C06372=1208.918,376.782,-77.823,-175.907,8.026,148.373
C06373=1208.922,376.534,-77.790,-175.909,8.024,148.372
C06374=1208.926,376.287,-77.756,-175.910,8.021,148.372
C06375=1208.931,376.039,-77.722,-175.911,8.018,148.372
C06376=1208.934,375.791,-77.688,-175.912,8.015,148.371
C06377=1208.939,375.544,-77.654,-175.913,8.012,148.371
C06378=1208.943,375.296,-77.620,-175.915,8.009,148.371
C06379=1208.947,375.049,-77.586,-175.915,8.006,148.370
C06380=1208.951,374.801,-77.553,-175.917,8.004,148.370
C06381=1208.955,374.553,-77.518,-175.918,8.000,148.369
C06382=1208.959,374.306,-77.485,-175.920,7.997,148.369
C06383=1208.963,374.058,-77.451,-175.921,7.994,148.368
C06384=1208.967,373.811,-77.418,-175.922,7.991,148.368
C06385=1208.971,373.563,-77.383,-175.923,7.989,148.368
C06386=1208.975,373.315,-77.350,-175.924,7.986,148.367
C06387=1208.979,373.067,-77.317,-175.926,7.983,148.367
C06388=1208.984,372.820,-77.282,-175.927,7.979,148.366
C06389=1208.988,372.572,-77.249,-175.929,7.977,148.366
C06390=1208.991,372.324,-77.215,-175.930,7.974,148.366
C06391=1208.995,372.076,-77.182,-175.931,7.971,148.365
C06392=1209.000,371.829,-77.147,-175.932,7.968,148.365
C06393=1209.004,371.581,-77.114,-175.934,7.964,148.364
C06394=1209.008,371.334,-77.081,-175.935,7.962,148.364
C06395=1209.012,371.086,-77.047,-175.936,7.959,148.364
C06396=1209.016,370.838,-77.013,-175.938,7.956,148.363
C06397=1209.021,370.590,-76.980,-175.939,7.953,148.363
C06398=1209.024,370.343,-76.946,-175.941,7.950,148.362
C06399=1209.029,370.095,-76.913,-175.942,7.947,148.362
C06400=1209.033,369.847,-76.880,-175.943,7.944,148.362
C06401=1209.037,369.599,-76.845,-175.945,7.941,148.361
C06402=1209.041,369.352,-76.812,-175.946,7.938,148.361
C06403=1209.045,369.104,-76.779,-175.948,7.935,148.360
C06404=1209.049,368.857,-76.745,-175.949,7.932,148.360
C06405=1209.053,368.609,-76.712,-175.950,7.929,148.360
C06406=1209.058,368.361,-76.678,-175.952,7.926,148.359
C06407=1209.062,368.113,-76.645,-175.953,7.923,148.359
C06408=1209.065,367.865,-76.610,-175.955,7.920,148.359
C06409=1209.069,367.618,-76.577,-175.956,7.917,148.358
C06410=1209.073,367.370,-76.544,-175.957,7.914,148.358
C06411=1209.079,367.090,-76.506,-175.959,7.910,148.357
C06412=1209.083,366.810,-76.468,-175.961,7.907,148.357
C06413=1209.087,366.529,-76.431,-175.963,7.904,148.357
C06414=1209.092,366.249,-76.393,-175.964,7.900,148.356
C06415=1209.097,366.001,-76.360,-175.966,7.898,148.356
C06416=1209.100,365.753,-76.326,-175.967,7.894,148.355
C06417=1209.104,365.506,-76.292,-175.969,7.892,148.355
C06418=1209.108,365.258,-76.259,-175.970,7.889,148.355
C06419=1209.112,365.010,-76.226,-175.972,7.885,148.354
C06420=1209.116,364.763,-76.193,-175.974,7.883,148.354
C06421=1209.120,364.515,-76.160,-175.975,7.879,148.354
C06422=1209.125,364.267,-76.126,-175.977,7.876,148.353
C06423=1209.129,364.019,-76.093,-175.978,7.874,148.353
C06424=1209.134,363.771,-76.060,-175.980,7.870,148.353
C06425=1209.138,363.524,-76.026,-175.981,7.867,148.352
C06426=1209.142,363.276,-75.993,-175.983,7.865,148.352
C06427=1209.146,363.029,-75.959,-175.985,7.861,148.352
C06428=1209.149,362.780,-75.926,-175.986,7.858,148.352
C06429=1209.153,362.533,-75.893,-175.988,7.855,148.351
C06430=1209.158,362.285,-75.860,-175.989,7.852,148.351
C06431=1209.162,362.037,-75.826,-175.991,7.849,148.351
C06432=1209.166,361.789,-75.793,-175.993,7.846,148.350
C06433=1209.170,361.542,-75.760,-175.994,7.843,148.350
C06434=1209.174,361.294,-75.727,-175.996,7.840,148.350
C06435=1209.178,361.046,-75.694,-175.998,7.837,148.349
C06436=1209.182,360.798,-75.661,-175.999,7.833,148.349
C06437=1209.186,360.551,-75.627,-176.001,7.831,148.349
C06438=1209.190,360.303,-75.596,-176.003,7.827,148.348
C06439=1209.194,360.055,-75.562,-176.004,7.825,148.348
C06440=1209.198,359.807,-75.529,-176.006,7.822,148.348
C06441=1209.203,359.559,-75.496,-176.008,7.819,148.348
C06442=1209.207,359.312,-75.463,-176.009,7.816,148.347
C06443=1209.211,359.064,-75.430,-176.011,7.813,148.347
C06444=1209.215,358.816,-75.397,-176.013,7.810,148.347
C06445=1209.219,358.569,-75.363,-176.015,7.806,148.346
C06446=1209.223,358.321,-75.330,-176.016,7.804,148.346
C06447=1209.228,358.072,-75.298,-176.018,7.800,148.346
C06448=1209.232,357.825,-75.265,-176.020,7.798,148.345
C06449=1209.235,357.577,-75.232,-176.022,7.794,148.345
C06450=1209.239,357.330,-75.199,-176.023,7.792,148.345
C06451=1209.244,357.082,-75.166,-176.025,7.788,148.345
C06452=1209.248,356.834,-75.133,-176.027,7.786,148.344
C06453=1209.252,356.586,-75.100,-176.029,7.782,148.344
C06454=1209.256,356.338,-75.067,-176.030,7.779,148.344
C06455=1209.260,356.090,-75.034,-176.033,7.776,148.344
C06456=1209.264,355.842,-75.002,-176.034,7.773,148.343
C06457=1209.268,355.595,-74.969,-176.036,7.770,148.343
C06458=1209.273,355.348,-74.936,-176.038,7.767,148.343
C06459=1209.277,355.100,-74.903,-176.039,7.764,148.342
C06460=1209.282,354.851,-74.871,-176.041,7.761,148.342
C06461=1209.285,354.604,-74.838,-176.043,7.758,148.342
C06462=1209.289,354.356,-74.805,-176.045,7.755,148.342
C06463=1209.294,354.108,-74.772,-176.047,7.752,148.341
C06464=1209.298,353.860,-74.739,-176.048,7.749,148.341
C06465=1209.302,353.613,-74.706,-176.051,7.746,148.341
C06466=1209.306,353.364,-74.674,-176.052,7.743,148.341
C06467=1209.310,353.117,-74.641,-176.054,7.740,148.340
C06468=1209.314,352.868,-74.609,-176.056,7.737,148.340
C06469=1209.319,352.621,-74.576,-176.058,7.734,148.340
C06470=1209.322,352.374,-74.543,-176.060,7.731,148.340
C06471=1209.327,352.126,-74.511,-176.062,7.728,148.339
C06472=1209.331,351.878,-74.478,-176.063,7.726,148.339
C06473=1209.335,351.630,-74.445,-176.065,7.722,148.339
C06474=1209.339,351.382,-74.413,-176.067,7.719,148.339
C06475=1209.343,351.134,-74.380,-176.069,7.716,148.338
C06476=1209.347,350.886,-74.347,-176.071,7.714,148.338
C06477=1209.352,350.639,-74.316,-176.073,7.710,148.338
C06478=1209.356,350.391,-74.282,-176.075,7.708,148.338
C06479=1209.360,350.143,-74.250,-176.077,7.704,148.338
C06480=1209.364,349.895,-74.217,-176.078,7.702,148.337
C06481=1209.368,349.647,-74.185,-176.080,7.698,148.337
C06482=1209.372,349.399,-74.152,-176.082,7.696,148.337
C06483=1209.376,349.152,-74.120,-176.084,7.692,148.337
C06484=1209.381,348.904,-74.087,-176.086,7.690,148.336
C06485=1209.385,348.656,-74.055,-176.088,7.686,148.336
C06486=1209.389,348.408,-74.023,-176.090,7.683,148.336
C06487=1209.393,348.160,-73.990,-176.092,7.681,148.336
C06488=1209.397,347.913,-73.958,-176.094,7.677,148.336
C06489=1209.401,347.665,-73.925,-176.096,7.675,148.335
C06490=1209.406,347.417,-73.893,-176.098,7.671,148.335
C06491=1209.409,347.168,-73.861,-176.099,7.669,148.335
C06492=1209.414,346.921,-73.828,-176.102,7.666,148.335
C06493=1209.418,346.673,-73.796,-176.103,7.663,148.335
C06494=1209.422,346.425,-73.764,-176.106,7.660,148.334
C06495=1209.427,346.177,-73.731,-176.107,7.657,148.334
C06496=1209.430,345.929,-73.699,-176.109,7.654,148.334
C06497=1209.435,345.681,-73.666,-176.111,7.651,148.334
C06498=1209.439,345.434,-73.635,-176.113,7.648,148.334
C06499=1209.443,345.186,-73.602,-176.115,7.645,148.333
C06500=1209.447,344.938,-73.570,-176.117,7.642,148.333
C06501=1209.451,344.689,-73.537,-176.119,7.639,148.333
C06502=1209.456,344.442,-73.506,-176.121,7.636,148.333
C06503=1209.460,344.194,-73.474,-176.123,7.633,148.333
C06504=1209.463,343.946,-73.441,-176.125,7.630,148.332
C06505=1209.468,343.699,-73.409,-176.127,7.627,148.332
C06506=1209.472,343.451,-73.377,-176.129,7.625,148.332
C06507=1209.477,343.202,-73.345,-176.131,7.621,148.332
C06508=1209.480,342.954,-73.313,-176.134,7.618,148.332
C06509=1209.485,342.707,-73.281,-176.135,7.616,148.332
C06510=1209.489,342.459,-73.248,-176.137,7.612,148.331
C06511=1209.493,342.211,-73.216,-176.139,7.610,148.331
C06512=1209.497,341.964,-73.184,-176.141,7.606,148.331
C06513=1209.501,341.716,-73.152,-176.143,7.604,148.331
C06514=1209.506,341.467,-73.120,-176.146,7.601,148.331
C06515=1209.511,341.189,-73.084,-176.148,7.597,148.330
C06516=1209.515,340.911,-73.049,-176.150,7.594,148.330
C06517=1209.520,340.633,-73.012,-176.152,7.591,148.330
C06518=1209.524,340.355,-72.977,-176.154,7.587,148.330
C06519=1209.529,340.107,-72.944,-176.157,7.585,148.330
C06520=1209.533,339.859,-72.913,-176.159,7.582,148.330
C06521=1209.537,339.611,-72.880,-176.161,7.579,148.329
C06522=1209.541,339.363,-72.848,-176.163,7.576,148.329
C06523=1209.545,339.116,-72.817,-176.165,7.573,148.329
C06524=1209.550,338.867,-72.785,-176.167,7.570,148.329
C06525=1209.553,338.619,-72.753,-176.169,7.567,148.329
C06526=1209.558,338.372,-72.721,-176.171,7.565,148.329
C06527=1209.562,338.124,-72.689,-176.173,7.562,148.329
C06528=1209.566,337.876,-72.657,-176.176,7.558,148.328
C06529=1209.571,337.628,-72.626,-176.177,7.556,148.328
C06530=1209.574,337.380,-72.594,-176.180,7.552,148.328
C06531=1209.579,337.131,-72.562,-176.182,7.550,148.328
C06532=1209.583,336.884,-72.530,-176.184,7.547,148.328
C06533=1209.587,336.636,-72.499,-176.186,7.544,148.328
C06534=1209.592,336.388,-72.466,-176.188,7.541,148.327
C06535=1209.595,336.140,-72.435,-176.190,7.538,148.327
C06536=1209.599,335.891,-72.403,-176.192,7.535,148.327
C06537=1209.604,335.644,-72.372,-176.194,7.532,148.327
C06538=1209.608,335.396,-72.340,-176.196,7.530,148.327
C06539=1209.613,335.148,-72.308,-176.199,7.526,148.327
C06540=1209.616,334.900,-72.276,-176.200,7.524,148.327
C06541=1209.620,334.652,-72.245,-176.203,7.521,148.327
C06542=1209.625,334.404,-72.214,-176.205,7.518,148.326
C06543=1209.629,334.156,-72.181,-176.207,7.515,148.326
C06544=1209.633,333.909,-72.150,-176.209,7.512,148.326
C06545=1209.637,333.660,-72.119,-176.211,7.510,148.326
C06546=1209.642,333.413,-72.087,-176.214,7.506,148.326
C06547=1209.645,333.165,-72.055,-176.215,7.504,148.326
C06548=1209.650,332.917,-72.025,-176.218,7.501,148.326
C06549=1209.654,332.668,-71.992,-176.220,7.498,148.326
C06550=1209.659,332.421,-71.961,-176.222,7.495,148.326
C06551=1209.663,332.172,-71.929,-176.225,7.492,148.326
C06552=1209.666,331.924,-71.898,-176.226,7.490,148.325
C06553=1209.671,331.677,-71.866,-176.228,7.486,148.325
C06554=1209.675,331.428,-71.835,-176.231,7.484,148.325
C06555=1209.679,331.181,-71.804,-176.233,7.481,148.325
C06556=1209.684,330.932,-71.772,-176.235,7.478,148.325
C06557=1209.688,330.685,-71.740,-176.237,7.475,148.325
C06558=1209.692,330.437,-71.708,-176.240,7.472,148.325
C06559=1209.696,330.189,-71.678,-176.241,7.470,148.325
C06560=1209.700,329.941,-71.646,-176.244,7.466,148.325
C06561=1209.705,329.693,-71.615,-176.246,7.464,148.324
C06562=1209.708,329.445,-71.583,-176.248,7.461,148.324
C06563=1209.713,329.197,-71.552,-176.251,7.458,148.324
C06564=1209.717,328.949,-71.521,-176.252,7.455,148.324
C06565=1209.721,328.701,-71.490,-176.255,7.452,148.324
C06566=1209.726,328.453,-71.458,-176.257,7.450,148.324
C06567=1209.730,328.205,-71.427,-176.259,7.446,148.324
C06568=1209.734,327.957,-71.397,-176.262,7.443,148.324
C06569=1209.738,327.709,-71.365,-176.264,7.441,148.324
C06570=1209.743,327.461,-71.334,-176.266,7.438,148.324
C06571=1209.746,327.213,-71.302,-176.268,7.435,148.324
C06572=1209.751,326.965,-71.271,-176.271,7.432,148.324
C06573=1209.755,326.717,-71.239,-176.272,7.430,148.323
C06574=1209.759,326.469,-71.209,-176.275,7.427,148.323
C06575=1209.764,326.221,-71.178,-176.277,7.423,148.323
C06576=1209.768,325.973,-71.146,-176.279,7.421,148.323
C06577=1209.772,325.725,-71.115,-176.282,7.418,148.323
C06578=1209.776,325.476,-71.084,-176.284,7.416,148.323
C06579=1209.780,325.229,-71.053,-176.286,7.413,148.323
C06580=1209.785,324.981,-71.022,-176.288,7.410,148.323
C06581=1209.789,324.732,-70.991,-176.291,7.407,148.323
C06582=1209.793,324.485,-70.961,-176.293,7.404,148.323
C06583=1209.797,324.237,-70.929,-176.295,7.402,148.323
C06584=1209.801,323.989,-70.898,-176.297,7.398,148.322
C06585=1209.806,323.741,-70.867,-176.299,7.396,148.322
C06586=1209.810,323.492,-70.836,-176.302,7.393,148.322
C06587=1209.814,323.245,-70.805,-176.304,7.390,148.322
C06588=1209.818,322.996,-70.774,-176.306,7.387,148.322
C06589=1209.822,322.748,-70.743,-176.309,7.384,148.322
C06590=1209.827,322.500,-70.713,-176.311,7.382,148.322
C06591=1209.831,322.252,-70.681,-176.313,7.379,148.322
C06592=1209.835,322.004,-70.650,-176.315,7.377,148.322
C06593=1209.840,321.756,-70.619,-176.318,7.373,148.322
C06594=1209.844,321.508,-70.588,-176.320,7.371,148.322
C06595=1209.848,321.260,-70.558,-176.322,7.368,148.322
C06596=1209.852,321.012,-70.527,-176.325,7.365,148.322
C06597=1209.856,320.763,-70.496,-176.327,7.362,148.322
C06598=1209.861,320.516,-70.465,-176.329,7.359,148.322
C06599=1209.865,320.268,-70.435,-176.331,7.357,148.322
C06600=1209.869,320.019,-70.404,-176.334,7.354,148.322
C06601=1209.873,319.771,-70.373,-176.336,7.352,148.322
C06602=1209.878,319.524,-70.342,-176.338,7.348,148.322
C06603=1209.881,319.276,-70.311,-176.341,7.345,148.322
C06604=1209.886,319.028,-70.280,-176.343,7.343,148.322
C06605=1209.890,318.780,-70.250,-176.345,7.340,148.321
C06606=1209.895,318.532,-70.219,-176.347,7.338,148.321
C06607=1209.898,318.283,-70.188,-176.350,7.334,148.321
C06608=1209.903,318.035,-70.158,-176.352,7.332,148.321
C06609=1209.908,317.787,-70.128,-176.354,7.329,148.321
C06610=1209.911,317.538,-70.097,-176.357,7.326,148.321
C06611=1209.915,317.290,-70.066,-176.359,7.324,148.321
C06612=1209.920,317.043,-70.035,-176.362,7.321,148.321
C06613=1209.924,316.795,-70.005,-176.363,7.318,148.321
C06614=1209.928,316.546,-69.974,-176.366,7.315,148.321
C06615=1209.933,316.298,-69.943,-176.368,7.313,148.321
C06616=1209.936,316.051,-69.913,-176.371,7.310,148.321
C06617=1209.941,315.803,-69.882,-176.373,7.307,148.321
C06618=1209.946,315.555,-69.852,-176.375,7.304,148.321
C06619=1209.949,315.278,-69.818,-176.378,7.301,148.321
C06620=1209.954,315.002,-69.784,-176.380,7.298,148.321
C06621=1209.959,314.726,-69.751,-176.383,7.295,148.321
C06622=1209.964,314.450,-69.716,-176.386,7.292,148.321
C06623=1209.969,314.202,-69.686,-176.389,7.289,148.321
C06624=1209.973,313.954,-69.656,-176.390,7.287,148.321
C06625=1209.977,313.706,-69.625,-176.393,7.284,148.321
C06626=1209.981,313.457,-69.595,-176.395,7.281,148.321
C06627=1209.985,313.209,-69.564,-176.398,7.278,148.321
C06628=1209.990,312.961,-69.535,-176.400,7.276,148.321
C06629=1209.994,312.713,-69.504,-176.402,7.273,148.321
C06630=1209.998,312.466,-69.474,-176.404,7.271,148.321
C06631=1210.003,312.217,-69.444,-176.407,7.268,148.321
C06632=1210.006,311.969,-69.413,-176.409,7.265,148.321
C06633=1210.011,311.721,-69.382,-176.412,7.262,148.321
C06634=1210.015,311.472,-69.353,-176.414,7.259,148.321
C06635=1210.020,311.224,-69.322,-176.416,7.257,148.321
C06636=1210.023,310.977,-69.292,-176.419,7.254,148.321
C06637=1210.028,310.728,-69.262,-176.421,7.252,148.321
C06638=1210.032,310.481,-69.232,-176.423,7.248,148.321
C06639=1210.037,310.231,-69.201,-176.426,7.246,148.321
C06640=1210.040,309.984,-69.171,-176.428,7.243,148.321
C06641=1210.045,309.736,-69.140,-176.431,7.240,148.321
C06642=1210.049,309.487,-69.111,-176.433,7.238,148.321
C06643=1210.054,309.239,-69.080,-176.436,7.235,148.321
C06644=1210.058,308.991,-69.051,-176.437,7.232,148.321
C06645=1210.062,308.744,-69.020,-176.440,7.229,148.321
C06646=1210.067,308.495,-68.990,-176.442,7.227,148.321
C06647=1210.071,308.247,-68.960,-176.445,7.224,148.321
C06648=1210.076,307.999,-68.930,-176.447,7.222,148.321
C06649=1210.079,307.750,-68.900,-176.450,7.219,148.321
C06650=1210.083,307.502,-68.870,-176.452,7.217,148.321
C06651=1210.088,307.254,-68.840,-176.454,7.214,148.321
C06652=1210.092,307.006,-68.810,-176.457,7.212,148.321
C06653=1210.097,306.757,-68.780,-176.459,7.208,148.321
C06654=1210.101,306.510,-68.750,-176.462,7.205,148.321
C06655=1210.105,306.261,-68.720,-176.464,7.203,148.321
C06656=1210.110,306.013,-68.690,-176.467,7.200,148.321
C06657=1210.114,305.765,-68.660,-176.469,7.198,148.321
C06658=1210.118,305.517,-68.631,-176.471,7.195,148.321
C06659=1210.122,305.269,-68.600,-176.474,7.193,148.321
C06660=1210.127,305.021,-68.570,-176.476,7.189,148.321
C06661=1210.131,304.772,-68.541,-176.478,7.187,148.321
C06662=1210.135,304.524,-68.512,-176.481,7.184,148.321
C06663=1210.140,304.276,-68.481,-176.483,7.182,148.321
C06664=1210.144,304.028,-68.451,-176.485,7.179,148.321
C06665=1210.148,303.780,-68.422,-176.488,7.177,148.321
C06666=1210.153,303.532,-68.391,-176.490,7.174,148.321
C06667=1210.157,303.283,-68.362,-176.492,7.172,148.321
C06668=1210.161,303.035,-68.332,-176.495,7.169,148.321
C06669=1210.165,302.787,-68.303,-176.498,7.165,148.321
C06670=1210.169,302.539,-68.273,-176.500,7.163,148.321
C06671=1210.174,302.291,-68.243,-176.503,7.160,148.321
C06672=1210.178,302.042,-68.213,-176.505,7.158,148.321
C06673=1210.182,301.794,-68.184,-176.507,7.155,148.321
C06674=1210.186,301.546,-68.154,-176.509,7.153,148.322
C06675=1210.191,301.298,-68.125,-176.512,7.150,148.322
C06676=1210.195,301.050,-68.094,-176.515,7.148,148.322
C06677=1210.199,300.801,-68.064,-176.517,7.145,148.322
C06678=1210.204,300.553,-68.035,-176.520,7.143,148.322
C06679=1210.208,300.305,-68.006,-176.522,7.140,148.322
C06680=1210.212,300.057,-67.976,-176.524,7.137,148.322
C06681=1210.217,299.809,-67.947,-176.527,7.134,148.322
C06682=1210.221,299.561,-67.918,-176.529,7.132,148.322
C06683=1210.226,299.312,-67.888,-176.532,7.129,148.322
C06684=1210.230,299.064,-67.858,-176.534,7.127,148.322
C06685=1210.234,298.816,-67.829,-176.537,7.124,148.322
C06686=1210.238,298.567,-67.799,-176.539,7.122,148.322
C06687=1210.243,298.319,-67.770,-176.541,7.119,148.322
C06688=1210.247,298.071,-67.740,-176.544,7.117,148.322
C06689=1210.251,297.823,-67.711,-176.546,7.113,148.322
C06690=1210.255,297.574,-67.681,-176.548,7.111,148.322
C06691=1210.259,297.326,-67.652,-176.551,7.108,148.322
C06692=1210.264,297.078,-67.623,-176.554,7.106,148.323
C06693=1210.268,296.830,-67.593,-176.556,7.103,148.323
C06694=1210.272,296.582,-67.564,-176.558,7.101,148.323
C06695=1210.277,296.334,-67.534,-176.561,7.098,148.323
C06696=1210.281,296.085,-67.505,-176.563,7.096,148.323
C06697=1210.285,295.837,-67.476,-176.566,7.093,148.323
C06698=1210.289,295.589,-67.446,-176.568,7.091,148.323
C06699=1210.294,295.341,-67.418,-176.571,7.088,148.323
C06700=1210.298,295.092,-67.388,-176.573,7.085,148.323
C06701=1210.303,294.844,-67.359,-176.576,7.083,148.323
C06702=1210.307,294.596,-67.329,-176.578,7.081,148.323
C06703=1210.311,294.348,-67.300,-176.581,7.078,148.323
C06704=1210.315,294.099,-67.270,-176.583,7.075,148.323
C06705=1210.320,293.851,-67.242,-176.586,7.072,148.323
C06706=1210.324,293.603,-67.213,-176.588,7.070,148.323
C06707=1210.329,293.355,-67.183,-176.590,7.067,148.323
C06708=1210.333,293.106,-67.154,-176.593,7.065,148.324
C06709=1210.337,292.857,-67.125,-176.595,7.063,148.324
C06710=1210.342,292.610,-67.096,-176.598,7.060,148.324
C06711=1210.346,292.362,-67.066,-176.600,7.058,148.324
C06712=1210.350,292.113,-67.037,-176.603,7.055,148.324
C06713=1210.354,291.865,-67.009,-176.605,7.053,148.324
C06714=1210.358,291.617,-66.979,-176.608,7.049,148.324
C06715=1210.363,291.369,-66.950,-176.610,7.048,148.324
C06716=1210.368,291.120,-66.922,-176.613,7.045,148.324
C06717=1210.372,290.872,-66.892,-176.615,7.042,148.324
C06718=1210.376,290.624,-66.863,-176.618,7.039,148.324
C06719=1210.381,290.375,-66.834,-176.620,7.037,148.324
C06720=1210.385,290.127,-66.805,-176.623,7.034,148.325
C06721=1210.389,289.879,-66.777,-176.625,7.032,148.325
C06722=1210.393,289.630,-66.747,-176.628,7.029,148.325
C06723=1210.398,289.356,-66.716,-176.630,7.027,148.325
C06724=1210.403,289.082,-66.683,-176.633,7.024,148.325
C06725=1210.407,288.808,-66.652,-176.636,7.021,148.325
C06726=1210.412,288.533,-66.620,-176.638,7.018,148.325
C06727=1210.416,288.285,-66.591,-176.641,7.016,148.325
C06728=1210.421,288.037,-66.562,-176.644,7.013,148.325
C06729=1210.426,287.789,-66.533,-176.646,7.011,148.326
C06730=1210.430,287.540,-66.504,-176.648,7.008,148.326
C06731=1210.434,287.293,-66.475,-176.651,7.006,148.326
C06732=1210.439,287.044,-66.447,-176.654,7.003,148.326
C06733=1210.443,286.795,-66.418,-176.656,7.001,148.326
C06734=1210.447,286.548,-66.389,-176.658,6.999,148.326
C06735=1210.452,286.299,-66.361,-176.661,6.996,148.326
C06736=1210.456,286.050,-66.331,-176.663,6.994,148.326
C06737=1210.461,285.802,-66.303,-176.666,6.991,148.326
C06738=1210.464,285.554,-66.274,-176.668,6.989,148.326
C06739=1210.469,285.305,-66.245,-176.671,6.986,148.326
C06740=1210.474,285.057,-66.217,-176.673,6.983,148.326
C06741=1210.477,284.809,-66.188,-176.676,6.982,148.327
C06742=1210.482,284.560,-66.159,-176.678,6.979,148.327
C06743=1210.487,284.312,-66.131,-176.680,6.976,148.327
C06744=1210.490,284.064,-66.102,-176.684,6.974,148.327
C06745=1210.495,283.816,-66.074,-176.686,6.971,148.327
C06746=1210.499,283.567,-66.046,-176.688,6.968,148.327
C06747=1210.504,283.319,-66.017,-176.690,6.966,148.327
C06748=1210.509,283.071,-65.988,-176.693,6.964,148.328
C06749=1210.512,282.822,-65.960,-176.696,6.961,148.328
C06750=1210.517,282.573,-65.931,-176.698,6.959,148.328
C06751=1210.521,282.326,-65.903,-176.701,6.956,148.328
C06752=1210.525,282.077,-65.874,-176.703,6.954,148.328
C06753=1210.530,281.829,-65.845,-176.705,6.952,148.328
C06754=1210.534,281.581,-65.817,-176.708,6.949,148.328
C06755=1210.539,281.332,-65.789,-176.711,6.947,148.328
C06756=1210.543,281.084,-65.761,-176.713,6.944,148.328
C06757=1210.547,280.836,-65.731,-176.715,6.942,148.328
C06758=1210.551,280.588,-65.703,-176.719,6.939,148.329
C06759=1210.556,280.339,-65.675,-176.721,6.937,148.329
C06760=1210.560,280.091,-65.647,-176.723,6.935,148.329
C06761=1210.565,279.842,-65.618,-176.726,6.932,148.329
C06762=1210.569,279.594,-65.590,-176.728,6.930,148.329
C06763=1210.574,279.345,-65.562,-176.731,6.927,148.329
C06764=1210.577,279.097,-65.534,-176.733,6.925,148.329
C06765=1210.582,278.848,-65.505,-176.736,6.923,148.330
C06766=1210.586,278.601,-65.476,-176.738,6.920,148.330
C06767=1210.591,278.352,-65.448,-176.740,6.918,148.330
C06768=1210.595,278.104,-65.420,-176.743,6.916,148.330
C06769=1210.600,277.856,-65.391,-176.746,6.913,148.330
C06770=1210.604,277.607,-65.363,-176.748,6.910,148.330
C06771=1210.608,277.359,-65.335,-176.751,6.908,148.330
C06772=1210.612,277.110,-65.307,-176.753,6.906,148.330
C06773=1210.617,276.862,-65.279,-176.755,6.903,148.330
C06774=1210.621,276.613,-65.250,-176.758,6.901,148.331
C06775=1210.626,276.366,-65.222,-176.761,6.899,148.331
C06776=1210.630,276.116,-65.195,-176.764,6.896,148.331
C06777=1210.635,275.868,-65.167,-176.766,6.894,148.331
C06778=1210.639,275.620,-65.139,-176.768,6.891,148.331
C06779=1210.644,275.371,-65.110,-176.771,6.889,148.331
C06780=1210.647,275.123,-65.082,-176.773,6.887,148.332
C06781=1210.652,274.875,-65.054,-176.775,6.884,148.332
C06782=1210.657,274.627,-65.026,-176.779,6.882,148.332
C06783=1210.661,274.378,-64.998,-176.781,6.879,148.332
C06784=1210.665,274.130,-64.970,-176.783,6.876,148.332
C06785=1210.670,273.881,-64.942,-176.786,6.875,148.332
C06786=1210.674,273.633,-64.914,-176.788,6.872,148.332
C06787=1210.678,273.384,-64.886,-176.791,6.870,148.333
C06788=1210.683,273.136,-64.858,-176.793,6.867,148.333
C06789=1210.687,272.888,-64.830,-176.796,6.865,148.333
C06790=1210.691,272.639,-64.802,-176.799,6.863,148.333
C06791=1210.696,272.391,-64.775,-176.801,6.860,148.333
C06792=1210.700,272.142,-64.746,-176.803,6.858,148.333
C06793=1210.704,271.895,-64.718,-176.806,6.855,148.333
C06794=1210.709,271.645,-64.691,-176.808,6.853,148.333
C06795=1210.713,271.397,-64.663,-176.811,6.851,148.334
C06796=1210.718,271.149,-64.635,-176.814,6.848,148.334
C06797=1210.722,270.900,-64.607,-176.816,6.847,148.334
C06798=1210.726,270.652,-64.579,-176.818,6.844,148.334
C06799=1210.731,270.404,-64.552,-176.821,6.841,148.334
C06800=1210.736,270.155,-64.524,-176.824,6.839,148.334
C06801=1210.740,269.907,-64.496,-176.826,6.837,148.335
C06802=1210.744,269.658,-64.468,-176.829,6.835,148.335
C06803=1210.748,269.410,-64.441,-176.831,6.832,148.335
C06804=1210.753,269.162,-64.413,-176.834,6.830,148.335
C06805=1210.757,268.913,-64.385,-176.836,6.827,148.335
C06806=1210.762,268.665,-64.357,-176.839,6.825,148.335
C06807=1210.766,268.417,-64.329,-176.841,6.823,148.336
C06808=1210.770,268.168,-64.302,-176.844,6.820,148.336
C06809=1210.775,267.920,-64.274,-176.846,6.818,148.336
C06810=1210.779,267.671,-64.247,-176.849,6.816,148.336
C06811=1210.783,267.423,-64.219,-176.852,6.814,148.336
C06812=1210.788,267.174,-64.192,-176.854,6.811,148.336
C06813=1210.793,266.926,-64.163,-176.857,6.810,148.337
C06814=1210.797,266.677,-64.136,-176.859,6.807,148.337
C06815=1210.801,266.429,-64.108,-176.861,6.804,148.337
C06816=1210.806,266.180,-64.081,-176.864,6.802,148.337
C06817=1210.810,265.932,-64.053,-176.867,6.799,148.337
C06818=1210.814,265.683,-64.026,-176.869,6.798,148.337
C06819=1210.819,265.435,-63.999,-176.871,6.795,148.338
C06820=1210.823,265.187,-63.971,-176.875,6.793,148.338
C06821=1210.828,264.938,-63.944,-176.877,6.790,148.338
C06822=1210.832,264.690,-63.916,-176.879,6.789,148.338
C06823=1210.836,264.441,-63.889,-176.881,6.786,148.338
C06824=1210.841,264.193,-63.862,-176.885,6.784,148.338
C06825=1210.845,263.945,-63.834,-176.887,6.782,148.339
C06826=1210.849,263.696,-63.807,-176.889,6.780,148.339
C06827=1210.855,263.423,-63.776,-176.892,6.777,148.339
C06828=1210.859,263.151,-63.746,-176.895,6.774,148.339
C06829=1210.864,262.878,-63.716,-176.898,6.772,148.339
C06830=1210.868,262.605,-63.686,-176.901,6.769,148.340
C06831=1210.873,262.357,-63.659,-176.903,6.767,148.340
C06832=1210.878,262.108,-63.632,-176.905,6.765,148.340
C06833=1210.882,261.860,-63.605,-176.908,6.762,148.340
C06834=1210.887,261.612,-63.577,-176.911,6.760,148.340
C06835=1210.891,261.363,-63.550,-176.913,6.758,148.341
C06836=1210.895,261.114,-63.523,-176.915,6.756,148.341
C06837=1210.900,260.866,-63.496,-176.919,6.753,148.341
C06838=1210.904,260.618,-63.468,-176.921,6.751,148.341
C06839=1210.909,260.369,-63.441,-176.923,6.749,148.341
C06840=1210.913,260.120,-63.413,-176.926,6.746,148.341
C06841=1210.918,259.872,-63.386,-176.929,6.744,148.342
C06842=1210.922,259.623,-63.360,-176.931,6.742,148.342
C06843=1210.926,259.375,-63.333,-176.933,6.740,148.342
C06844=1210.931,259.127,-63.305,-176.936,6.737,148.342
C06845=1210.935,258.879,-63.278,-176.939,6.735,148.342
C06846=1210.939,258.629,-63.250,-176.941,6.733,148.342
C06847=1210.944,258.381,-63.223,-176.943,6.731,148.343
C06848=1210.949,258.132,-63.196,-176.946,6.728,148.343
C06849=1210.953,257.884,-63.170,-176.949,6.727,148.343
C06850=1210.957,257.636,-63.143,-176.951,6.724,148.343
C06851=1210.962,257.387,-63.116,-176.954,6.723,148.343
C06852=1210.967,257.139,-63.089,-176.957,6.720,148.344
C06853=1210.971,256.889,-63.061,-176.959,6.718,148.344
C06854=1210.974,256.641,-63.035,-176.961,6.716,148.344
C06855=1210.979,256.393,-63.008,-176.964,6.714,148.344
C06856=1210.984,256.144,-62.981,-176.967,6.711,148.344
C06857=1210.988,255.896,-62.954,-176.969,6.709,148.345
C06858=1210.992,255.648,-62.927,-176.972,6.707,148.345
C06859=1210.997,255.399,-62.900,-176.974,6.705,148.345
C06860=1211.002,255.151,-62.873,-176.977,6.702,148.345
C06861=1211.006,254.902,-62.846,-176.979,6.700,148.346
C06862=1211.010,254.654,-62.819,-176.982,6.698,148.346
C06863=1211.015,254.405,-62.792,-176.984,6.696,148.346
C06864=1211.019,254.156,-62.765,-176.987,6.693,148.346
C06865=1211.024,253.908,-62.738,-176.990,6.691,148.346
C06866=1211.028,253.660,-62.711,-176.992,6.689,148.346
C06867=1211.033,253.410,-62.685,-176.994,6.687,148.347
C06868=1211.037,253.162,-62.658,-176.997,6.685,148.347
C06869=1211.041,252.914,-62.632,-177.000,6.682,148.347
C06870=1211.046,252.665,-62.605,-177.002,6.680,148.347
C06871=1211.050,252.417,-62.577,-177.004,6.678,148.347
C06872=1211.054,252.169,-62.551,-177.007,6.676,148.348
C06873=1211.059,251.919,-62.525,-177.010,6.674,148.348
C06874=1211.064,251.671,-62.498,-177.012,6.671,148.348
C06875=1211.068,251.423,-62.471,-177.015,6.670,148.348
C06876=1211.073,251.174,-62.444,-177.017,6.667,148.349
C06877=1211.077,250.925,-62.418,-177.020,6.666,148.349
C06878=1211.081,250.677,-62.391,-177.022,6.663,148.349
C06879=1211.086,250.429,-62.364,-177.025,6.661,148.349
C06880=1211.090,250.180,-62.338,-177.028,6.659,148.349
C06881=1211.095,249.931,-62.311,-177.030,6.657,148.350
C06882=1211.099,249.683,-62.285,-177.032,6.655,148.350
C06883=1211.104,249.435,-62.258,-177.036,6.652,148.350
C06884=1211.108,249.186,-62.232,-177.038,6.650,148.350
C06885=1211.112,248.937,-62.205,-177.040,6.648,148.351
C06886=1211.117,248.689,-62.178,-177.042,6.646,148.351
C06887=1211.121,248.440,-62.152,-177.045,6.644,148.351
C06888=1211.126,248.191,-62.125,-177.048,6.641,148.351
C06889=1211.130,247.943,-62.099,-177.050,6.639,148.351
C06890=1211.135,247.694,-62.072,-177.053,6.637,148.352
C06891=1211.139,247.446,-62.046,-177.055,6.635,148.352
C06892=1211.144,247.197,-62.020,-177.058,6.633,148.352
C06893=1211.148,246.949,-61.993,-177.060,6.631,148.352
C06894=1211.153,246.700,-61.967,-177.063,6.628,148.352
C06895=1211.157,246.452,-61.941,-177.066,6.626,148.353
C06896=1211.162,246.204,-61.914,-177.068,6.625,148.353
C06897=1211.166,245.955,-61.888,-177.071,6.622,148.353
C06898=1211.171,245.706,-61.861,-177.073,6.621,148.353
C06899=1211.175,245.457,-61.835,-177.076,6.618,148.354
C06900=1211.179,245.209,-61.809,-177.078,6.616,148.354
C06901=1211.184,244.960,-61.782,-177.081,6.614,148.354
C06902=1211.188,244.712,-61.756,-177.084,6.612,148.354
C06903=1211.193,244.463,-61.729,-177.086,6.610,148.355
C06904=1211.197,244.214,-61.704,-177.088,6.608,148.355
C06905=1211.202,243.966,-61.677,-177.092,6.605,148.355
C06906=1211.206,243.717,-61.651,-177.094,6.603,148.355
C06907=1211.210,243.469,-61.625,-177.096,6.601,148.356
C06908=1211.215,243.220,-61.598,-177.099,6.599,148.356
C06909=1211.219,242.971,-61.573,-177.101,6.597,148.356
C06910=1211.223,242.723,-61.546,-177.104,6.595,148.356
C06911=1211.228,242.474,-61.520,-177.107,6.593,148.357
C06912=1211.233,242.227,-61.494,-177.109,6.590,148.357
C06913=1211.237,241.978,-61.468,-177.112,6.589,148.357
C06914=1211.242,241.729,-61.442,-177.114,6.587,148.357
C06915=1211.246,241.480,-61.415,-177.117,6.585,148.357
C06916=1211.250,241.232,-61.389,-177.119,6.583,148.358
C06917=1211.255,240.983,-61.363,-177.122,6.581,148.358
C06918=1211.260,240.734,-61.338,-177.125,6.578,148.358
C06919=1211.264,240.486,-61.311,-177.127,6.576,148.358
C06920=1211.269,240.237,-61.285,-177.130,6.574,148.359
C06921=1211.273,239.988,-61.259,-177.132,6.572,148.359
C06922=1211.277,239.740,-61.233,-177.135,6.570,148.359
C06923=1211.282,239.492,-61.207,-177.137,6.568,148.359
C06924=1211.287,239.243,-61.181,-177.139,6.566,148.360
C06925=1211.291,238.994,-61.155,-177.142,6.564,148.360
C06926=1211.295,238.745,-61.129,-177.145,6.562,148.360
C06927=1211.299,238.496,-61.104,-177.148,6.560,148.360
C06928=1211.305,238.249,-61.077,-177.150,6.557,148.361
C06929=1211.309,238.000,-61.051,-177.153,6.556,148.361
C06930=1211.313,237.751,-61.025,-177.155,6.554,148.361
C06931=1211.318,237.479,-60.997,-177.158,6.551,148.361
C06932=1211.323,237.209,-60.969,-177.160,6.549,148.362
C06933=1211.328,236.937,-60.941,-177.163,6.547,148.362
C06934=1211.334,236.665,-60.913,-177.166,6.544,148.362
C06935=1211.338,236.416,-60.887,-177.169,6.543,148.362
C06936=1211.342,236.168,-60.861,-177.172,6.541,148.363
C06937=1211.346,235.919,-60.835,-177.174,6.538,148.363
C06938=1211.351,235.671,-60.809,-177.176,6.537,148.363
C06939=1211.355,235.423,-60.784,-177.179,6.535,148.364
C06940=1211.359,235.174,-60.758,-177.182,6.533,148.364
C06941=1211.364,234.925,-60.732,-177.184,6.530,148.364
C06942=1211.369,234.676,-60.706,-177.187,6.528,148.364
C06943=1211.373,234.428,-60.680,-177.190,6.526,148.365
C06944=1211.377,234.179,-60.655,-177.192,6.524,148.365
C06945=1211.382,233.931,-60.629,-177.194,6.522,148.365
C06946=1211.386,233.682,-60.604,-177.197,6.520,148.365
C06947=1211.391,233.433,-60.578,-177.200,6.518,148.366
C06948=1211.396,233.185,-60.552,-177.202,6.516,148.366
C06949=1211.400,232.936,-60.527,-177.204,6.514,148.366
C06950=1211.404,232.687,-60.502,-177.207,6.513,148.366
C06951=1211.410,232.438,-60.476,-177.210,6.510,148.367
C06952=1211.414,232.190,-60.450,-177.212,6.508,148.367
C06953=1211.418,231.941,-60.424,-177.215,6.506,148.367
C06954=1211.423,231.693,-60.399,-177.218,6.504,148.367
C06955=1211.427,231.444,-60.373,-177.220,6.502,148.368
C06956=1211.432,231.195,-60.347,-177.223,6.500,148.368
C06957=1211.436,230.947,-60.322,-177.225,6.498,148.368
C06958=1211.441,230.698,-60.297,-177.228,6.496,148.368
C06959=1211.445,230.449,-60.271,-177.230,6.494,148.369
C06960=1211.450,230.201,-60.246,-177.233,6.493,148.369
C06961=1211.454,229.952,-60.220,-177.235,6.490,148.369
C06962=1211.459,229.704,-60.195,-177.238,6.489,148.369
C06963=1211.464,229.454,-60.169,-177.241,6.486,148.370
C06964=1211.468,229.206,-60.144,-177.243,6.484,148.370
C06965=1211.472,228.958,-60.119,-177.246,6.482,148.370
C06966=1211.476,228.709,-60.093,-177.248,6.480,148.371
C06967=1211.481,228.460,-60.069,-177.251,6.478,148.371
C06968=1211.485,228.211,-60.043,-177.254,6.476,148.371
C06969=1211.490,227.963,-60.017,-177.256,6.474,148.372
C06970=1211.495,227.714,-59.992,-177.258,6.472,148.372
C06971=1211.499,227.465,-59.967,-177.261,6.470,148.372
C06972=1211.504,227.217,-59.941,-177.264,6.469,148.372
C06973=1211.508,226.968,-59.916,-177.266,6.467,148.373
C06974=1211.513,226.719,-59.890,-177.269,6.465,148.373
C06975=1211.517,226.471,-59.865,-177.271,6.463,148.373
C06976=1211.521,226.222,-59.841,-177.274,6.461,148.373
C06977=1211.526,225.973,-59.815,-177.277,6.458,148.374
C06978=1211.530,225.725,-59.789,-177.279,6.456,148.374
C06979=1211.535,225.476,-59.765,-177.282,6.455,148.374
C06980=1211.540,225.227,-59.739,-177.285,6.453,148.375
C06981=1211.545,224.978,-59.714,-177.287,6.451,148.375
C06982=1211.549,224.730,-59.689,-177.290,6.449,148.375
C06983=1211.553,224.481,-59.665,-177.292,6.447,148.375
C06984=1211.558,224.232,-59.639,-177.295,6.445,148.376
C06985=1211.563,223.984,-59.614,-177.297,6.443,148.376
C06986=1211.567,223.735,-59.588,-177.300,6.441,148.376
C06987=1211.572,223.487,-59.563,-177.302,6.439,148.376
C06988=1211.576,223.238,-59.539,-177.305,6.437,148.377
C06989=1211.581,222.989,-59.514,-177.307,6.435,148.377
C06990=1211.585,222.740,-59.488,-177.310,6.434,148.377
C06991=1211.590,222.491,-59.463,-177.313,6.432,148.378
C06992=1211.594,222.243,-59.438,-177.315,6.430,148.378
C06993=1211.599,221.994,-59.414,-177.318,6.428,148.378
C06994=1211.603,221.745,-59.388,-177.320,6.426,148.379
C06995=1211.608,221.497,-59.363,-177.323,6.424,148.379
C06996=1211.612,221.248,-59.338,-177.325,6.422,148.379
C06997=1211.617,220.999,-59.313,-177.328,6.420,148.380
C06998=1211.621,220.750,-59.288,-177.331,6.418,148.380
C06999=1211.625,220.502,-59.264,-177.333,6.415,148.380
C07000=1211.630,220.253,-59.239,-177.336,6.414,148.380
C07001=1211.635,220.004,-59.214,-177.339,6.412,148.381
C07002=1211.639,219.756,-59.189,-177.341,6.410,148.381
C07003=1211.644,219.507,-59.164,-177.344,6.408,148.381
C07004=1211.649,219.258,-59.139,-177.347,6.406,148.382
C07005=1211.652,219.010,-59.114,-177.349,6.404,148.382
C07006=1211.657,218.761,-59.090,-177.351,6.402,148.382
C07007=1211.662,218.511,-59.065,-177.354,6.400,148.382
C07008=1211.666,218.264,-59.040,-177.357,6.399,148.383
C07009=1211.671,218.015,-59.015,-177.359,6.397,148.383
C07010=1211.676,217.765,-58.990,-177.362,6.395,148.383
C07011=1211.680,217.517,-58.966,-177.365,6.393,148.384
C07012=1211.684,217.268,-58.940,-177.367,6.391,148.384
C07013=1211.689,217.020,-58.916,-177.370,6.389,148.384
C07014=1211.694,216.771,-58.891,-177.372,6.388,148.385
C07015=1211.698,216.522,-58.867,-177.375,6.385,148.385
C07016=1211.703,216.273,-58.842,-177.377,6.383,148.385
C07017=1211.708,216.025,-58.818,-177.380,6.382,148.385
C07018=1211.711,215.776,-58.793,-177.383,6.380,148.386
C07019=1211.716,215.527,-58.768,-177.385,6.378,148.386
C07020=1211.720,215.278,-58.743,-177.388,6.376,148.386
C07021=1211.725,215.030,-58.719,-177.390,6.374,148.387
C07022=1211.730,214.781,-58.695,-177.393,6.372,148.387
C07023=1211.734,214.532,-58.670,-177.396,6.371,148.387
C07024=1211.739,214.283,-58.646,-177.398,6.369,148.388
C07025=1211.744,214.035,-58.621,-177.401,6.367,148.388
C07026=1211.747,213.786,-58.596,-177.403,6.365,148.388
C07027=1211.752,213.537,-58.571,-177.406,6.363,148.389
C07028=1211.757,213.289,-58.547,-177.408,6.361,148.389
C07029=1211.762,213.040,-58.522,-177.411,6.359,148.389
C07030=1211.766,212.791,-58.498,-177.414,6.357,148.390
C07031=1211.771,212.542,-58.473,-177.416,6.356,148.390
C07032=1211.775,212.294,-58.449,-177.419,6.354,148.390
C07033=1211.780,212.045,-58.424,-177.422,6.352,148.391
C07034=1211.784,211.796,-58.400,-177.424,6.350,148.391
C07035=1211.790,211.525,-58.374,-177.427,6.348,148.391
C07036=1211.795,211.255,-58.347,-177.430,6.346,148.392
C07037=1211.799,210.984,-58.320,-177.433,6.344,148.392
C07038=1211.804,210.714,-58.294,-177.435,6.342,148.392
C07039=1211.809,210.466,-58.269,-177.438,6.340,148.393
C07040=1211.813,210.217,-58.245,-177.441,6.338,148.393
C07041=1211.818,209.967,-58.221,-177.443,6.336,148.393
C07042=1211.823,209.719,-58.197,-177.446,6.334,148.394
C07043=1211.827,209.470,-58.173,-177.449,6.333,148.394
C07044=1211.832,209.222,-58.148,-177.451,6.331,148.394
C07045=1211.836,208.973,-58.124,-177.454,6.329,148.395
C07046=1211.840,208.724,-58.100,-177.457,6.327,148.395
C07047=1211.845,208.475,-58.075,-177.459,6.325,148.395
C07048=1211.850,208.226,-58.052,-177.461,6.323,148.395
C07049=1211.854,207.978,-58.028,-177.464,6.321,148.396
C07050=1211.859,207.729,-58.003,-177.467,6.319,148.396
C07051=1211.863,207.480,-57.979,-177.469,6.318,148.396
C07052=1211.868,207.232,-57.954,-177.472,6.316,148.397
C07053=1211.873,206.982,-57.930,-177.475,6.314,148.397
C07054=1211.878,206.734,-57.906,-177.477,6.312,148.397
C07055=1211.881,206.485,-57.882,-177.480,6.310,148.398
C07056=1211.887,206.236,-57.857,-177.482,6.309,148.398
C07057=1211.891,205.987,-57.834,-177.485,6.307,148.398
C07058=1211.896,205.739,-57.810,-177.487,6.306,148.399
C07059=1211.900,205.490,-57.786,-177.490,6.304,148.399
C07060=1211.905,205.240,-57.761,-177.493,6.302,148.399
C07061=1211.909,204.992,-57.737,-177.495,6.300,148.400
C07062=1211.914,204.743,-57.713,-177.498,6.298,148.400
C07063=1211.918,204.495,-57.689,-177.500,6.296,148.400
C07064=1211.923,204.246,-57.666,-177.503,6.295,148.401
C07065=1211.928,203.997,-57.641,-177.506,6.293,148.401
C07066=1211.932,203.748,-57.617,-177.508,6.291,148.401
C07067=1211.936,203.499,-57.593,-177.511,6.289,148.402
C07068=1211.941,203.251,-57.569,-177.514,6.287,148.402
C07069=1211.945,203.002,-57.546,-177.516,6.285,148.402
C07070=1211.951,202.753,-57.521,-177.519,6.284,148.403
C07071=1211.955,202.504,-57.498,-177.522,6.282,148.403
C07072=1211.960,202.255,-57.474,-177.524,6.281,148.404
C07073=1211.964,202.007,-57.450,-177.526,6.279,148.404
C07074=1211.968,201.757,-57.426,-177.529,6.277,148.404
C07075=1211.973,201.509,-57.402,-177.532,6.275,148.405
C07076=1211.977,201.260,-57.379,-177.534,6.273,148.405
C07077=1211.982,201.011,-57.354,-177.537,6.272,148.405
C07078=1211.987,200.762,-57.331,-177.540,6.270,148.406
C07079=1211.992,200.514,-57.307,-177.542,6.268,148.406
C07080=1211.996,200.265,-57.283,-177.545,6.266,148.406
C07081=1212.001,200.016,-57.259,-177.547,6.264,148.407
C07082=1212.005,199.767,-57.236,-177.550,6.262,148.407
C07083=1212.010,199.518,-57.212,-177.553,6.261,148.407
C07084=1212.014,199.270,-57.188,-177.555,6.260,148.408
C07085=1212.019,199.021,-57.165,-177.558,6.258,148.408
C07086=1212.023,198.772,-57.141,-177.560,6.256,148.408
C07087=1212.028,198.523,-57.118,-177.563,6.254,148.409
C07088=1212.032,198.274,-57.093,-177.565,6.252,148.409
C07089=1212.037,198.025,-57.070,-177.568,6.250,148.409
C07090=1212.041,197.776,-57.046,-177.571,6.249,148.410
C07091=1212.047,197.527,-57.022,-177.573,6.247,148.410
C07092=1212.051,197.278,-56.998,-177.576,6.245,148.410
C07093=1212.056,197.029,-56.975,-177.579,6.243,148.411
C07094=1212.060,196.781,-56.951,-177.581,6.242,148.411
C07095=1212.065,196.532,-56.928,-177.583,6.240,148.412
C07096=1212.070,196.283,-56.904,-177.586,6.238,148.412
C07097=1212.073,196.035,-56.881,-177.589,6.237,148.412
C07098=1212.078,195.786,-56.857,-177.591,6.235,148.413
C07099=1212.083,195.537,-56.834,-177.594,6.233,148.413
C07100=1212.087,195.288,-56.811,-177.597,6.231,148.413
C07101=1212.092,195.039,-56.787,-177.599,6.229,148.414
C07102=1212.097,194.790,-56.763,-177.601,6.228,148.414
C07103=1212.101,194.541,-56.740,-177.604,6.226,148.414
C07104=1212.106,194.292,-56.716,-177.607,6.225,148.415
C07105=1212.111,194.043,-56.693,-177.609,6.223,148.415
C07106=1212.115,193.795,-56.669,-177.612,6.221,148.415
C07107=1212.120,193.546,-56.646,-177.615,6.219,148.416
C07108=1212.125,193.297,-56.623,-177.617,6.217,148.416
C07109=1212.130,193.048,-56.599,-177.620,6.216,148.416
C07110=1212.134,192.799,-56.576,-177.622,6.215,148.417
C07111=1212.138,192.551,-56.553,-177.625,6.213,148.417
C07112=1212.143,192.302,-56.529,-177.627,6.211,148.417
C07113=1212.148,192.053,-56.506,-177.630,6.209,148.418
C07114=1212.152,191.804,-56.482,-177.633,6.208,148.418
C07115=1212.157,191.555,-56.459,-177.636,6.206,148.419
C07116=1212.162,191.306,-56.436,-177.638,6.204,148.419
C07117=1212.166,191.057,-56.412,-177.641,6.203,148.419
C07118=1212.170,190.808,-56.390,-177.643,6.201,148.420
C07119=1212.175,190.559,-56.366,-177.646,6.199,148.420
C07120=1212.180,190.311,-56.343,-177.648,6.197,148.420
C07121=1212.185,190.062,-56.320,-177.651,6.196,148.421
C07122=1212.190,189.813,-56.297,-177.654,6.194,148.421
C07123=1212.194,189.564,-56.274,-177.656,6.193,148.422
C07124=1212.198,189.315,-56.250,-177.659,6.191,148.422
C07125=1212.203,189.066,-56.227,-177.661,6.189,148.422
C07126=1212.208,188.817,-56.204,-177.664,6.187,148.423
C07127=1212.212,188.568,-56.180,-177.666,6.185,148.423
C07128=1212.216,188.319,-56.158,-177.669,6.184,148.423
C07129=1212.222,188.071,-56.135,-177.672,6.183,148.424
C07130=1212.226,187.822,-56.111,-177.674,6.181,148.424
C07131=1212.231,187.573,-56.088,-177.677,6.179,148.425
C07132=1212.235,187.324,-56.065,-177.680,6.178,148.425
C07133=1212.240,187.075,-56.042,-177.682,6.176,148.425
C07134=1212.244,186.826,-56.018,-177.685,6.174,148.426
C07135=1212.249,186.578,-55.996,-177.687,6.173,148.426
C07136=1212.254,186.329,-55.973,-177.690,6.171,148.426
C07137=1212.259,186.079,-55.950,-177.692,6.169,148.427
C07138=1212.263,185.830,-55.927,-177.695,6.167,148.427
C07139=1212.268,185.561,-55.902,-177.698,6.166,148.428
C07140=1212.273,185.291,-55.877,-177.701,6.164,148.428
C07141=1212.278,185.022,-55.852,-177.703,6.162,148.428
C07142=1212.283,184.753,-55.827,-177.706,6.160,148.429
C07143=1212.288,184.503,-55.804,-177.709,6.159,148.429
C07144=1212.292,184.254,-55.782,-177.712,6.157,148.430
C07145=1212.297,184.006,-55.759,-177.714,6.156,148.430
C07146=1212.302,183.757,-55.735,-177.717,6.154,148.430
C07147=1212.306,183.508,-55.712,-177.719,6.152,148.431
C07148=1212.311,183.258,-55.690,-177.722,6.151,148.431
C07149=1212.315,183.010,-55.667,-177.725,6.149,148.431
C07150=1212.320,182.761,-55.644,-177.727,6.148,148.432
C07151=1212.325,182.512,-55.621,-177.729,6.146,148.432
C07152=1212.329,182.263,-55.599,-177.732,6.144,148.433
C07153=1212.334,182.014,-55.575,-177.735,6.143,148.433
C07154=1212.338,181.766,-55.553,-177.738,6.141,148.433
C07155=1212.343,181.516,-55.530,-177.740,6.140,148.434
C07156=1212.347,181.268,-55.507,-177.743,6.138,148.434
C07157=1212.352,181.019,-55.484,-177.745,6.136,148.435
C07158=1212.357,180.770,-55.462,-177.748,6.134,148.435
C07159=1212.362,180.521,-55.439,-177.751,6.133,148.435
C07160=1212.366,180.272,-55.417,-177.753,6.132,148.436
C07161=1212.371,180.023,-55.394,-177.756,6.130,148.436
C07162=1212.376,179.774,-55.371,-177.758,6.128,148.437
C07163=1212.380,179.525,-55.349,-177.761,6.127,148.437
C07164=1212.385,179.276,-55.325,-177.763,6.126,148.437
C07165=1212.390,179.027,-55.304,-177.766,6.124,148.438
C07166=1212.394,178.778,-55.281,-177.768,6.122,148.438
C07167=1212.399,178.529,-55.258,-177.771,6.120,148.438
C07168=1212.403,178.281,-55.236,-177.774,6.119,148.439
C07169=1212.408,178.032,-55.212,-177.776,6.118,148.439
C07170=1212.412,177.782,-55.190,-177.779,6.116,148.440
C07171=1212.417,177.534,-55.167,-177.782,6.114,148.440
C07172=1212.422,177.285,-55.145,-177.784,6.112,148.440
C07173=1212.426,177.036,-55.122,-177.786,6.111,148.441
C07174=1212.431,176.787,-55.100,-177.789,6.109,148.441
C07175=1212.436,176.537,-55.078,-177.792,6.108,148.442
C07176=1212.440,176.289,-55.055,-177.795,6.106,148.442
C07177=1212.445,176.040,-55.033,-177.797,6.105,148.443
C07178=1212.450,175.791,-55.010,-177.800,6.103,148.443
C07179=1212.454,175.542,-54.988,-177.802,6.101,148.443
C07180=1212.459,175.293,-54.965,-177.805,6.100,148.444
C07181=1212.464,175.044,-54.943,-177.808,6.099,148.444
C07182=1212.469,174.795,-54.921,-177.810,6.097,148.445
C07183=1212.473,174.546,-54.898,-177.813,6.095,148.445
C07184=1212.478,174.297,-54.876,-177.816,6.093,148.445
C07185=1212.482,174.049,-54.853,-177.818,6.092,148.446
C07186=1212.487,173.799,-54.831,-177.820,6.091,148.446
C07187=1212.492,173.551,-54.809,-177.823,6.089,148.447
C07188=1212.496,173.302,-54.786,-177.826,6.087,148.447
C07189=1212.501,173.052,-54.764,-177.828,6.086,148.447
C07190=1212.506,172.804,-54.742,-177.831,6.085,148.448
C07191=1212.510,172.554,-54.720,-177.834,6.083,148.448
C07192=1212.515,172.306,-54.697,-177.836,6.082,148.448
C07193=1212.520,172.057,-54.675,-177.839,6.080,148.449
C07194=1212.524,171.807,-54.653,-177.841,6.078,148.449
C07195=1212.528,171.559,-54.630,-177.844,6.077,148.450
C07196=1212.533,171.310,-54.608,-177.846,6.076,148.450
C07197=1212.538,171.061,-54.586,-177.849,6.074,148.451
C07198=1212.543,170.812,-54.564,-177.852,6.072,148.451
C07199=1212.548,170.563,-54.542,-177.854,6.071,148.452
C07200=1212.552,170.314,-54.519,-177.857,6.070,148.452
C07201=1212.557,170.065,-54.497,-177.859,6.068,148.452
C07202=1212.561,169.816,-54.475,-177.862,6.066,148.453
C07203=1212.566,169.567,-54.453,-177.864,6.065,148.453
C07204=1212.571,169.318,-54.431,-177.867,6.064,148.454
C07205=1212.575,169.069,-54.408,-177.870,6.062,148.454
C07206=1212.580,168.820,-54.386,-177.872,6.061,148.454
C07207=1212.584,168.571,-54.364,-177.875,6.059,148.455
C07208=1212.590,168.322,-54.342,-177.878,6.057,148.455
C07209=1212.594,168.073,-54.320,-177.881,6.056,148.456
C07210=1212.599,167.824,-54.298,-177.883,6.055,148.456
C07211=1212.603,167.575,-54.276,-177.885,6.053,148.456
C07212=1212.608,167.326,-54.255,-177.888,6.051,148.457
C07213=1212.612,167.077,-54.233,-177.891,6.050,148.457
C07214=1212.618,166.828,-54.210,-177.893,6.049,148.458
C07215=1212.622,166.578,-54.188,-177.896,6.047,148.458
C07216=1212.627,166.330,-54.167,-177.898,6.046,148.458
C07217=1212.632,166.082,-54.144,-177.901,6.044,148.459
C07218=1212.636,165.832,-54.122,-177.904,6.042,148.459
C07219=1212.641,165.584,-54.100,-177.906,6.041,148.460
C07220=1212.645,165.334,-54.078,-177.909,6.040,148.460
C07221=1212.650,165.086,-54.057,-177.911,6.038,148.461
C07222=1212.654,164.836,-54.035,-177.914,6.037,148.461
C07223=1212.659,164.587,-54.014,-177.917,6.035,148.462
C07224=1212.664,164.338,-53.991,-177.919,6.034,148.462
C07225=1212.669,164.089,-53.969,-177.922,6.032,148.462
C07226=1212.674,163.840,-53.947,-177.924,6.031,148.463
C07227=1212.678,163.591,-53.926,-177.927,6.029,148.463
C07228=1212.683,163.342,-53.904,-177.930,6.028,148.464
C07229=1212.688,163.093,-53.882,-177.932,6.027,148.464
C07230=1212.693,162.844,-53.860,-177.935,6.025,148.464
C07231=1212.697,162.595,-53.838,-177.938,6.023,148.465
C07232=1212.702,162.346,-53.816,-177.940,6.022,148.465
C07233=1212.707,162.098,-53.795,-177.942,6.020,148.466
C07234=1212.711,161.848,-53.773,-177.945,6.019,148.466
C07235=1212.716,161.599,-53.752,-177.948,6.018,148.467
C07236=1212.720,161.350,-53.730,-177.950,6.016,148.467
C07237=1212.725,161.101,-53.708,-177.952,6.015,148.467
C07238=1212.730,160.852,-53.686,-177.955,6.013,148.468
C07239=1212.734,160.603,-53.664,-177.958,6.012,148.468
C07240=1212.739,160.354,-53.643,-177.960,6.011,148.469
C07241=1212.744,160.105,-53.622,-177.963,6.009,148.469
C07242=1212.749,159.856,-53.600,-177.966,6.007,148.470
C07243=1212.753,159.587,-53.577,-177.969,6.006,148.470
C07244=1212.758,159.318,-53.553,-177.971,6.005,148.471
C07245=1212.763,159.049,-53.530,-177.974,6.003,148.471
C07246=1212.769,158.780,-53.507,-177.977,6.002,148.472
C07247=1212.774,158.531,-53.485,-177.979,6.000,148.472
C07248=1212.778,158.282,-53.463,-177.982,5.999,148.473
C07249=1212.783,158.032,-53.442,-177.985,5.997,148.473
C07250=1212.788,157.784,-53.420,-177.987,5.996,148.473
C07251=1212.793,157.535,-53.399,-177.990,5.995,148.474
C07252=1212.797,157.286,-53.378,-177.993,5.993,148.474
C07253=1212.801,157.037,-53.356,-177.995,5.991,148.475
C07254=1212.806,156.788,-53.334,-177.997,5.990,148.475
C07255=1212.811,156.538,-53.313,-178.001,5.989,148.476
C07256=1212.816,156.290,-53.291,-178.003,5.988,148.476
C07257=1212.821,156.041,-53.270,-178.005,5.986,148.476
C07258=1212.825,155.791,-53.248,-178.008,5.984,148.477
C07259=1212.829,155.543,-53.227,-178.011,5.984,148.477
C07260=1212.835,155.293,-53.206,-178.013,5.982,148.478
C07261=1212.839,155.045,-53.185,-178.016,5.980,148.478
C07262=1212.844,154.795,-53.163,-178.019,5.979,148.479
C07263=1212.849,154.546,-53.142,-178.021,5.978,148.479
C07264=1212.854,154.298,-53.120,-178.023,5.977,148.479
C07265=1212.858,154.048,-53.099,-178.026,5.975,148.480
C07266=1212.862,153.799,-53.078,-178.029,5.973,148.480
C07267=1212.868,153.550,-53.057,-178.031,5.972,148.481
C07268=1212.872,153.301,-53.035,-178.034,5.971,148.481
C07269=1212.877,153.052,-53.015,-178.037,5.970,148.482
C07270=1212.881,152.803,-52.993,-178.039,5.968,148.482
C07271=1212.886,152.554,-52.972,-178.042,5.966,148.483
C07272=1212.891,152.305,-52.950,-178.044,5.966,148.483
C07273=1212.896,152.056,-52.929,-178.047,5.964,148.484
C07274=1212.900,151.807,-52.907,-178.049,5.963,148.484
C07275=1212.905,151.558,-52.886,-178.052,5.961,148.484
C07276=1212.910,151.308,-52.866,-178.055,5.960,148.485
C07277=1212.914,151.060,-52.844,-178.057,5.959,148.485
C07278=1212.920,150.811,-52.823,-178.060,5.957,148.486
C07279=1212.924,150.561,-52.801,-178.062,5.956,148.486
C07280=1212.928,150.313,-52.781,-178.065,5.954,148.487
C07281=1212.933,150.063,-52.760,-178.068,5.953,148.487
C07282=1212.938,149.815,-52.738,-178.070,5.952,148.488
C07283=1212.943,149.566,-52.718,-178.073,5.950,148.488
C07284=1212.947,149.316,-52.697,-178.075,5.949,148.489
C07285=1212.952,149.067,-52.675,-178.078,5.948,148.489
C07286=1212.957,148.818,-52.655,-178.080,5.947,148.490
C07287=1212.962,148.569,-52.634,-178.083,5.945,148.490
C07288=1212.967,148.320,-52.612,-178.086,5.944,148.490
C07289=1212.971,148.071,-52.592,-178.088,5.943,148.491
C07290=1212.976,147.821,-52.570,-178.091,5.941,148.491
C07291=1212.981,147.573,-52.549,-178.094,5.940,148.492
C07292=1212.985,147.324,-52.528,-178.096,5.938,148.492
C07293=1212.990,147.074,-52.507,-178.098,5.937,148.493
C07294=1212.995,146.826,-52.487,-178.102,5.936,148.493
C07295=1212.999,146.577,-52.465,-178.104,5.934,148.494
C07296=1213.005,146.328,-52.444,-178.106,5.933,148.494
C07297=1213.008,146.078,-52.423,-178.110,5.932,148.495
